    //Calculate Stop TIME (Start TIME + Shift Length TIME)
    IF  OEE_SP.Length.CurrentTime.wDay = 0 THEN			// When Length Day = 0, Stop Time Calculcation is Different because TimeStruct has a minimum of 1 for Days
    	_Year_Month_Day_TS[0].wHour 	 := OEE_SP.Length.CurrentTime.wHour;
    	_Year_Month_Day_TS[0].wMinute 	 := OEE_SP.Length.CurrentTime.wMinute;
    	_Stop_Time_DW 					 := ((_Start_Time_DW+_Year_Month_Day_DW[0])-_Year_Month_Day_DW[1]);	// Add Shift Length Time to Start Time and subtract Year/Month/Day = Stop Time
    	_Stop_Time_DT 					 := DWORD_TO_DT(_Stop_Time_DW);										// Convert Stop Time fron DWORD to DATE_AND_TIME format	
    	OEE_SP.Stop.CurrentTime 		 := DT_TO_SYSTEMTIME(_Stop_Time_DT);								// Convert Stop Time from DATE_AND_TIME format to TIMESTRUCT
    ELSE                                                                                
    	_Stop_Time_DW 					:= (_Start_Time_DW+_Length_Time_DW)-_Year_Month_Day_DW[1];	// Add Shift Length Time to Start Time and subtract Year/Month = Stop Time
    	_Stop_Time_DT 					:= DWORD_TO_DT(_Stop_Time_DW);								// Convert Stop Time fron DWORD to DATE_AND_TIME format
    	OEE_SP.Stop.CurrentTime 		:= DT_TO_SYSTEMTIME(_Stop_Time_DT);							// Convert Stop Time from DATE_AND_TIME format to TIMESTRUCT
    	OEE_SP.Stop.CurrentTime.wDay 	:= OEE_SP.Stop.CurrentTime.wDay + 1;
    END_IF
	
	IF NOT OEE_SP.Break_Active AND OEE_SP.Active THEN
		_fb_MachinePerfomance(Perf := OEE_SP.MachinePerformance, Control := Control, Data_Reset := _Mach_Perf_Reset);
	END_IF
    //--------------------------------------------------------Availability---------------------------------------------------------
    
    //Calculate total time the machine has been avaliable to run (i.e. operators not on a break)
    IF  OEE_SP.Active AND NOT OEE_SP.Break_Active AND Control.SystemTime.SecondPulse THEN;
    	OEE_SP.Production_Seconds := OEE_SP.Production_Seconds + 1;
    END_IF
    _Production_Time_T := REAL_TO_TIME(OEE_SP.Production_Seconds)*1000;
    _Production_Time_DT := TIME_TO_DT(_Production_Time_T);
    _Production_Time_TS := DT_TO_SYSTEMTIME(_Production_Time_DT);
    IF OEE_SP.Production_Seconds < 86400 THEN
    	OEE_SP.Production_Time.CurrentTime := _Production_Time_TS;
    	OEE_SP.Production_Time.CurrentTime.wDay := 0;
    ELSE
    	OEE_SP.Production_Time.CurrentTime := _Production_Time_TS;
    	OEE_SP.Production_Time.CurrentTime.wDay := _Production_Time_TS.wDay-1;
    END_IF	
    
    //Calculate the time the machine has been producing
    IF OEE_SP.Active AND NOT OEE_SP.Break_Active AND Control.SystemTime.SecondPulse AND (Control.PackMLState.Execute OR Control.PackMLState.Suspended OR Control.PackMLState.Suspending OR Control.PackMLState.UnSuspending) THEN;
    	OEE_SP.Operating_Seconds := OEE_SP.Operating_Seconds + 1;
    END_IF
    
    _Operating_Time_T := REAL_TO_TIME(OEE_SP.Operating_Seconds)*1000;
    _Operating_Time_DT := TIME_TO_DT(_Operating_Time_T);
    _Operating_Time_TS := DT_TO_SYSTEMTIME(_Operating_Time_DT);
    IF OEE_SP.Operating_Seconds < 86400 THEN
    	OEE_SP.Operating_Time.CurrentTime := (_Operating_Time_TS);
    	OEE_SP.Operating_Time.CurrentTime.wDay := 0;
    ELSE
    	OEE_SP.Operating_Time.CurrentTime := (_Operating_Time_TS);
    	OEE_SP.Operating_Time.CurrentTime.wDay := _Operating_Time_TS.wDay-1;
    END_IF
    
    //Calculate Break Time
    IF OEE_SP.Active AND OEE_SP.Break_Active AND Control.SystemTime.SecondPulse THEN;
    	OEE_SP.Break_Seconds := OEE_SP.Break_Seconds + 1; 
    END_IF
    _Break_Time_T := LREAL_TO_TIME(OEE_SP.Break_Seconds)*1000;
    _Break_Time_DT := TIME_TO_DT(_Break_Time_T);
    _Break_Time_TS := DT_TO_SYSTEMTIME(_Break_Time_DT);
    IF OEE_SP.Break_Seconds < 86400 THEN
    	OEE_SP.Break_Time.CurrentTime := (_Break_Time_TS);
    	OEE_SP.Break_Time.CurrentTime.wDay := 0;
    ELSE
    	OEE_SP.Break_Time.CurrentTime := (_Break_Time_TS);
    	OEE_SP.Break_Time.CurrentTime.wDay := _Break_Time_TS.wDay-1;
    END_IF
     
    //Calculate Avaliability
    IF (OEE_SP.Operating_Seconds > 0 AND OEE_SP.Production_Seconds > 0.0) AND Control.SystemTime.SecondPulse THEN;
    	OEE_SP.Availability := ((OEE_SP.Operating_Seconds/ F_CheckDivReal(OEE_SP.Production_Seconds))*100);
    ELSIF (OEE_SP.Operating_Seconds <= 0 OR OEE_SP.Production_Seconds <= 0.0) THEN;
    	OEE_SP.Availability := 0.0;
    END_IF
    
    //--------------------------------------------------------Performance---------------------------------------------------------
    
    //Calculate Performance
    IF (OEE_SP.TotalPieces > 0 AND OEE_SP.Operating_Seconds > 0.0 AND OEE_SP.TargetRate > 0.0) AND Control.SystemTime.SecondPulse  THEN;
    	OEE_SP.Performance := DINT_TO_REAL(OEE_SP.TotalPieces)/OEE_SP.Operating_Seconds/(F_CheckDivReal(OEE_SP.TargetRate/60))*100;
    ELSIF ((OEE_SP.TotalPieces <= 0) OR (OEE_SP.Operating_Seconds <= 0.0) OR (OEE_SP.TargetRate <= 0.0)) THEN;
    	OEE_SP.Performance := 0;
    ELSIF OEE_SP.Performance > 100.0 THEN;
    	OEE_SP.Performance := 100;
    END_IF
    
    //--------------------------------------------------------Quality---------------------------------------------------------
    
    //Calculate Quality
    IF (OEE_SP.GoodPieces > 0 AND OEE_SP.TotalPieces > 0) AND Control.SystemTime.SecondPulse  THEN;
    	OEE_SP.Quality := DINT_TO_REAL(OEE_SP.GoodPieces)/DINT_TO_REAL(F_CheckDivDint(OEE_SP.TotalPieces))*100;
    ELSIF (OEE_SP.GoodPieces <= 0 OR OEE_SP.TotalPieces <= 0) THEN;
    	OEE_SP.Quality := 0.0;
    END_IF
    //--------------------------------------------------------------OEE-----------------------------------------------------------------
    
    //Calculate OEE 
    IF Control.SystemTime.SecondPulse THEN
    OEE_SP.OEE := ((OEE_SP.Availability/100) * (OEE_SP.Performance/100) * (OEE_SP.Quality/100)) *100;
    IF OEE_SP.OEE >100.0 THEN
    	OEE_SP.OEE:=100;
    END_IF
    END_IF
    //--------------------------------------------------------Supply Availability---------------------------------------------------------
    
    //Calculate Infeed Supply
    IF (OEE_SP.Operating_Seconds > 0 AND OEE_SP.Production_Seconds > 0.0) AND Control.SystemTime.SecondPulse  THEN;
    	OEE_SP.SupplyAvaliability := ((OEE_SP.Operating_Seconds-(OEE_SP.SupplyDownTime_Seconds))/F_CheckDivReal(OEE_SP.Operating_Seconds)*100);
    ELSIF (OEE_SP.Operating_Seconds <= 0 OR OEE_SP.Production_Seconds <= 0.0) THEN;
    	OEE_SP.SupplyAvaliability := 0.0;
    END_IF
    //--------------------------------------------------------Outfeed Availability---------------------------------------------------------
    //Calculate Outfeed Availability
    IF (OEE_SP.Operating_Seconds > 0 AND OEE_SP.Production_Seconds > 0.0) AND Control.SystemTime.SecondPulse  THEN;
    	OEE_SP.OutfeedAvaliability := ((OEE_SP.Operating_Seconds-(OEE_SP.OutfeedDownTime_Seconds))/F_CheckDivReal(OEE_SP.Operating_Seconds)*100);
    ELSIF (OEE_SP.Operating_Seconds <= 0 OR OEE_SP.Production_Seconds <= 0.0) THEN;
    	OEE_SP.OutfeedAvaliability := 0.0;
    END_IF
    //--------------------------------------------------------Total Pieces---------------------------------------------------------
    OEE_SP.TotalPieces := (OEE_SP.GoodPieces + OEE_SP.RejectPieces);
    OEE.Outputs.Availability := OEE_SP.Availability;
    OEE.Outputs.Performance := OEE_SP.Performance;
    OEE.Outputs.Quality:= OEE_SP.Quality;
    OEE.Outputs.OEE:= OEE_SP.OEE;
	
	 //--------------------------------------------------------Active Shift---------------------------------------------------------
    _Current_Time_DT := SYSTEMTIME_TO_DT(_Current_Time.CurrentTime);
    _Current_Time_DW	:=DT_TO_DWORD(_Current_Time_DT);
    
    IF ((_Current_Time_DW > _Start_Time_DW) AND (_Current_Time_DW <= _Stop_Time_DW)) THEN //OR (REAL_TO_UDINT(OEE_SP.Production_Seconds) < (_Stop_Time_DW - _Start_Time_DW)) THEN
    	OEE.Outputs.Active := TRUE;
    	OEE_SP.Active := TRUE;
    ELSE 
    	OEE.Outputs.Active := FALSE;
    	OEE_SP.Active := FALSE;
    END_IF

	IF OEE.Inputs.Break_Active AND OEE.Outputs.Active THEN
		OEE_SP.Break_Active:=TRUE;
	ELSE 
		OEE_SP.Break_Active:=FALSE;
	END_IF
	
	OEE_SP.StateCurrent := Control.PackMLState.CurrentState;

END_FUNCTION_BLOCK

// Objects/FB_PML_V4_01/FB_PackML
FUNCTION_BLOCK FINAL FB_PackML
VAR_IN_OUT
	PackML							: ST_PMLData;
	Control							: ST_System;
END_VAR
VAR
	_Cfg_ModeTransitions			: ARRAY[0..9, 0..31] OF BOOL;
	_Index							: INT;
	_LastState						: DINT;
	_LastUnit						: DINT;
	_MessageClearPointer			: INT;
	_WarningRefreshPointer			: INT;
	_WarningRefresh					: F_TRIG;
END_VAR
VAR CONSTANT
	_MaxModeLength					: INT := 7;
	_MaxStateLength					: INT := 17;
END_VAR
VAR PERSISTENT
	_LS_H_IndicatorMatrix				: ARRAY[0..31] OF DINT :=[1032,33792,1032,361504,66784,361504,198690,67616,1028,1028,1032,99360,1216,82984,295936,1032,1028];
	_PB_IndicatorMatrix					: ARRAY[0..31] OF DINT :=[0,256,32768,0,32768,32768,32768,16384,0,256,0,0,32768,32768,16384,32768,256,0];			
	_LS_H_IndicatorDescription			: ARRAY[0..31] OF STRING(40) := ['','Alarm','Abnormal Stop','Controlled Stop','','Alert','Starved Upstream','Blocked Downstream','','','Low Material','Material Exhausted','','','Alert','Alarm','Starting / Restarting','','','','','','','','','','','','',''];		
	_PB_IndicatorDescription			: ARRAY[0..31] OF STRING(40) := ['','','','','','','','','Ready to Reset','','','','','','Ready to Start','Running','','','','','','','','','','','','','','','',''];		
END_VAR

M_Administration();
M_Commands();
M_Indicators();
M_ModeControl();
M_SafetyBreach();
M_StateMapping();
M_StateTransitions();
M_TransitionCounts();

METHOD PRIVATE M_Administration
VAR_INPUT
END_VAR
VAR_INST
	_index					: INT;
END_VAR
IF PackML.Status.UnitModeCurrent > _maxModeLength THEN
	PackML.Control.UnitMode := 0;
	PackML.Status.UnitModeCurrent := 0;
END_IF

//Time spent in Mode
//The elapsed time the machine has spent in that mode since it entered that mode.  Array index is equal to designation of the mode.
IF PackML.Status.UnitModeChangeInProcess THEN
	PackML.Admin.ModeCurrentTime[PackML.Status.UnitModeCurrent] := 0;
END_IF
IF Control.SystemTime.SecondPulse THEN
	PackML.Admin.ModeCurrentTime[PackML.Status.UnitModeCurrent] := PackML.Admin.ModeCurrentTime[PackML.Status.UnitModeCurrent] + 1;
	IF PackML.Admin.ModeCurrentTime[PackML.Status.UnitModeCurrent] < 0 THEN
		PackML.Admin.ModeCurrentTime[PackML.Status.UnitModeCurrent] := 0;
	END_IF
	IF PackML.Admin.ResetTimerCounters THEN
		FOR _index := 0 TO _maxModeLength DO
			PackML.Admin.ModeCurrentTime[_index] := 0;
		END_FOR
	END_IF
END_IF

//Cumulative TIME In Each Mode
//The cumulative elapsed time the machine has spent in each mode since it’s timers and counters were reset.  
IF Control.SystemTime.SecondPulse THEN
	PackML.Admin.ModeCummulativeTime[PackML.Status.UnitModeCurrent] := PackML.Admin.ModeCummulativeTime[PackML.Status.UnitModeCurrent] + 1;
	IF PackML.Admin.ModeCummulativeTime[PackML.Status.UnitModeCurrent] < 0 THEN
		PackML.Admin.ModeCummulativeTime[PackML.Status.UnitModeCurrent] := 0;
	END_IF
	IF PackML.Admin.ResetTimerCounters THEN
		FOR _index := 0 TO _maxModeLength DO
			PackML.Admin.ModeCummulativeTime[_index] := 0;
		END_FOR
	END_IF
END_IF

//TIME spent in State
//The elapsed time the machine has spent in that State since it entered that State.  Array index is equal to designation of the mode.
IF PackML.Status.StateChangeInProgress THEN
	PackML.Admin.StateCurrentTime[PackML.Status.UnitModeCurrent,PackML.Status.StateCurrent] := 0;
END_IF
IF Control.SystemTime.SecondPulse THEN
	PackML.Admin.StateCurrentTime[PackML.Status.UnitModeCurrent,PackML.Status.StateCurrent] := PackML.Admin.StateCurrentTime[PackML.Status.UnitModeCurrent,PackML.Status.StateCurrent] + 1;
	IF PackML.Admin.StateCurrentTime[PackML.Status.UnitModeCurrent,PackML.Status.StateCurrent] < 0 THEN
		PackML.Admin.StateCurrentTime[PackML.Status.UnitModeCurrent,PackML.Status.StateCurrent] := 0;
	END_IF
	IF PackML.Admin.ResetTimerCounters THEN
		FOR _index := 0 TO _maxStateLength DO
			PackML.Admin.StateCurrentTime[PackML.Status.UnitModeCurrent,_index] := 0;
		END_FOR
	END_IF
END_IF

//Cumulative Time In Each Mode
//The cumulative elapsed time the machine has spent in each mode since it’s timers and counters were reset.  
IF Control.SystemTime.SecondPulse THEN
	PackML.Admin.StateCummulativeTime[PackML.Status.UnitModeCurrent,PackML.Status.StateCurrent] := PackML.Admin.StateCummulativeTime[PackML.Status.UnitModeCurrent,PackML.Status.StateCurrent] + 1;
	IF PackML.Admin.StateCummulativeTime[PackML.Status.UnitModeCurrent,PackML.Status.StateCurrent] < 0 THEN
		PackML.Admin.StateCummulativeTime[PackML.Status.UnitModeCurrent,PackML.Status.StateCurrent] := 0;
	END_IF
	IF PackML.Admin.ResetTimerCounters THEN
		FOR _index := 0 TO _maxStateLength DO
			PackML.Admin.StateCummulativeTime[PackML.Status.UnitModeCurrent,_index] := 0;
		END_FOR
	END_IF
END_IF
END_METHOD

METHOD PRIVATE M_Commands
VAR_INPUT
END_VAR
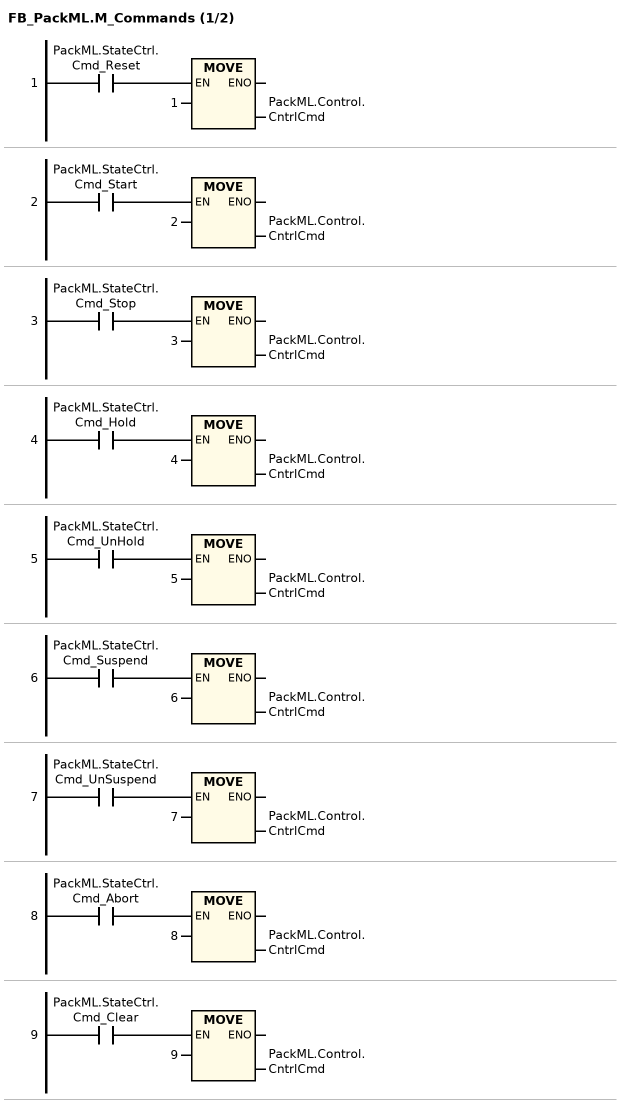
// NETWORK 1
IF PackML.StateCtrl.Cmd_Reset THEN PackML.Control.CntrlCmd := 1; END_IF

// NETWORK 2
IF PackML.StateCtrl.Cmd_Start THEN PackML.Control.CntrlCmd := 2; END_IF

// NETWORK 3
IF PackML.StateCtrl.Cmd_Stop THEN PackML.Control.CntrlCmd := 3; END_IF

// NETWORK 4
IF PackML.StateCtrl.Cmd_Hold THEN PackML.Control.CntrlCmd := 4; END_IF

// NETWORK 5
IF PackML.StateCtrl.Cmd_UnHold THEN PackML.Control.CntrlCmd := 5; END_IF

// NETWORK 6
IF PackML.StateCtrl.Cmd_Suspend THEN PackML.Control.CntrlCmd := 6; END_IF

// NETWORK 7
IF PackML.StateCtrl.Cmd_UnSuspend THEN PackML.Control.CntrlCmd := 7; END_IF

// NETWORK 8
IF PackML.StateCtrl.Cmd_Abort THEN PackML.Control.CntrlCmd := 8; END_IF

// NETWORK 9
IF PackML.StateCtrl.Cmd_Clear THEN PackML.Control.CntrlCmd := 9; END_IF

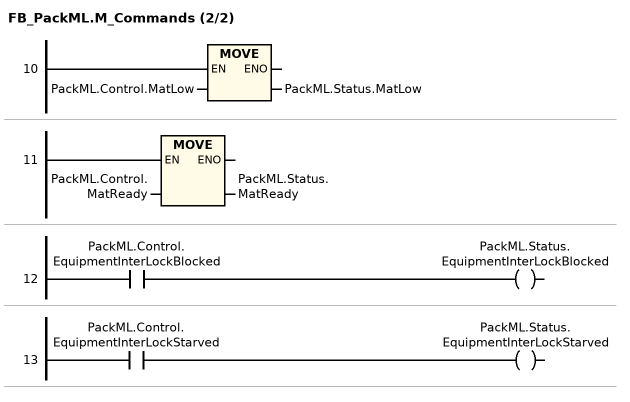
// NETWORK 10
PackML.Status.MatLow := PackML.Control.MatLow;

// NETWORK 11
PackML.Status.MatReady := PackML.Control.MatReady;

// NETWORK 12
PackML.Status.EquipmentInterLockBlocked := PackML.Control.EquipmentInterLockBlocked;

// NETWORK 13
PackML.Status.EquipmentInterLockStarved := PackML.Control.EquipmentInterLockStarved;
END_METHOD

METHOD PRIVATE M_Indicators
VAR_INST
	_i 		: DINT;
	_f_trig	: F_TRIG;
	_r_trig	: R_TRIG;
	k : bool;
END_VAR
PackML.Indicator.LS_H_Output := _LS_H_IndicatorMatrix[PackML.Status.StateCurrent];

//Red Lamp
IF PackML.Indicator.LS_H_Output.0 THEN
	PackML.Indicator.RedLamp := Control.SystemTime.PulseFlash;
ELSIF PackML.Indicator.LS_H_Output.1 AND Control.Outputs.Alarm THEN
	PackML.Indicator.RedLamp := Control.SystemTime.FastFlash;
ELSIF PackML.Indicator.LS_H_Output.2 THEN
	PackML.Indicator.RedLamp := Control.SystemTime.SlowFlash;
ELSIF PackML.Indicator.LS_H_Output.3 THEN
	PackML.Indicator.RedLamp := TRUE;
ELSE
	PackML.Indicator.RedLamp := FALSE;
END_IF

//Amber Lamp
IF PackML.Indicator.LS_H_Output.4 THEN
	PackML.Indicator.AmberLamp := Control.SystemTime.PulseFlash;
ELSIF PackML.Indicator.LS_H_Output.5 AND Control.Outputs.Alert THEN
	PackML.Indicator.AmberLamp := Control.SystemTime.FastFlash;
ELSIF PackML.Indicator.LS_H_Output.6 THEN
	PackML.Indicator.AmberLamp := Control.SystemTime.SlowFlash;
ELSIF PackML.Indicator.LS_H_Output.7 THEN
	PackML.Indicator.AmberLamp := TRUE;
ELSE
	PackML.Indicator.AmberLamp := FALSE;
END_IF

//Blue Lamp
IF PackML.Indicator.LS_H_Output.8 THEN
	PackML.Indicator.BlueLamp := Control.SystemTime.PulseFlash;
ELSIF PackML.Indicator.LS_H_Output.9 THEN
	PackML.Indicator.BlueLamp := Control.SystemTime.FastFlash;
ELSIF PackML.Indicator.LS_H_Output.10 THEN
	FOR	_i := 0 TO SIZEOF(Packml.Status.MatLow) BY 1 DO
		IF Packml.Status.MatLow[_i] THEN
			PackML.Indicator.BlueLamp := Control.SystemTime.SlowFlash;
			EXIT;
		END_IF
	END_FOR
ELSIF PackML.Indicator.LS_H_Output.11 THEN
	FOR	_i := 0 TO SIZEOF(Packml.Status.MatReady) BY 1 DO
		_f_trig(CLK:= Packml.Status.MatReady[_i]);
		IF _f_trig.Q THEN
			PackML.Indicator.BlueLamp := TRUE;
			EXIT;
		END_IF
		_r_trig(CLK:= Packml.Status.MatReady[_i]);
		IF _r_trig.Q THEN
			PackML.Indicator.BlueLamp := FALSE;
			EXIT;
		END_IF
	END_FOR
ELSE
	PackML.Indicator.BlueLamp := FALSE;
END_IF

//Green Lamp
IF PackML.Indicator.LS_H_Output.12 THEN
	PackML.Indicator.GreenLamp := Control.SystemTime.PulseFlash;
ELSIF PackML.Indicator.LS_H_Output.13 THEN
	PackML.Indicator.GreenLamp := Control.SystemTime.FastFlash;
ELSIF PackML.Indicator.LS_H_Output.14 THEN
	PackML.Indicator.GreenLamp := Control.SystemTime.SlowFlash;
ELSIF PackML.Indicator.LS_H_Output.15 THEN
	PackML.Indicator.GreenLamp := TRUE;
ELSE
	PackML.Indicator.GreenLamp := FALSE;
END_IF

//Horn
IF PackML.Indicator.LS_H_Output.16 AND Control.Outputs.Alert THEN
	PackML.Indicator.Horn := Control.SystemTime.PulseFlash;
ELSIF PackML.Indicator.LS_H_Output.17 AND Control.Outputs.Alarm THEN
	PackML.Indicator.Horn := Control.SystemTime.FastFlash;
ELSIF PackML.Indicator.LS_H_Output.18 THEN
	PackML.Indicator.Horn := Control.SystemTime.SlowFlash;
ELSIF PackML.Indicator.LS_H_Output.19 THEN
	PackML.Indicator.Horn := TRUE;
ELSE
	PackML.Indicator.Horn := FALSE;
END_IF

PackML.Indicator.PB_Output := _PB_IndicatorMatrix[PackML.Status.StateCurrent];

//Red Button
IF PackML.Indicator.PB_Output.0 THEN
	PackML.Indicator.RedButton := Control.SystemTime.PulseFlash;
ELSIF PackML.Indicator.PB_Output.1 THEN
	PackML.Indicator.RedButton := Control.SystemTime.FastFlash;
ELSIF PackML.Indicator.PB_Output.2 THEN
	PackML.Indicator.RedButton := Control.SystemTime.SlowFlash;
ELSIF PackML.Indicator.PB_Output.3 THEN
	PackML.Indicator.RedButton := TRUE;
ELSE
	PackML.Indicator.RedButton := FALSE;
END_IF

//Amber Button
IF PackML.Indicator.PB_Output.4 THEN
	PackML.Indicator.AmberButton := Control.SystemTime.PulseFlash;
ELSIF PackML.Indicator.PB_Output.5 THEN
	PackML.Indicator.AmberButton := Control.SystemTime.FastFlash;
ELSIF PackML.Indicator.PB_Output.6 THEN
	PackML.Indicator.AmberButton := Control.SystemTime.SlowFlash;
ELSIF PackML.Indicator.PB_Output.7 THEN
	PackML.Indicator.AmberButton := TRUE;
ELSE
	PackML.Indicator.AmberButton := FALSE;
END_IF

//Blue Button
IF PackML.Indicator.PB_Output.8 THEN
	PackML.Indicator.BlueButton := Control.SystemTime.PulseFlash;
ELSIF PackML.Indicator.PB_Output.9 THEN
	PackML.Indicator.BlueButton := Control.SystemTime.FastFlash;
ELSIF PackML.Indicator.PB_Output.10 THEN
	PackML.Indicator.BlueButton := Control.SystemTime.SlowFlash;
ELSIF PackML.Indicator.PB_Output.11 THEN
	PackML.Indicator.BlueButton := TRUE;
ELSE
	PackML.Indicator.BlueButton := FALSE;
END_IF

//Green Button
IF PackML.Indicator.PB_Output.12 THEN
	PackML.Indicator.GreenButton := Control.SystemTime.PulseFlash;
ELSIF PackML.Indicator.PB_Output.13 THEN
	PackML.Indicator.GreenButton := Control.SystemTime.FastFlash;
ELSIF PackML.Indicator.PB_Output.14 THEN
	PackML.Indicator.GreenButton := Control.SystemTime.SlowFlash;
ELSIF PackML.Indicator.PB_Output.15 THEN
	PackML.Indicator.GreenButton := TRUE;
ELSE
	PackML.Indicator.GreenButton := FALSE;
END_IF
END_METHOD

METHOD PRIVATE M_ModeControl
VAR_INPUT
END_VAR
VAR_INST
END_VAR
IF Control.SystemTime.FirstCycle THEN
	FOR _index := 0 TO 9 BY 1 DO
		_cfg_ModeTransitions[_index,2] := TRUE;
		_cfg_ModeTransitions[_index,9] := TRUE;
	END_FOR
END_IF

IF PackML.Control.UnitMode >= 1 AND PackML.Control.UnitMode <= 32 AND (PackML.Control.UnitMode <> PackML.Status.UnitModeCurrent) THEN
	IF _cfg_ModeTransitions[PackML.Status.UnitModeCurrent,PackML.Status.StateCurrent] AND _cfg_ModeTransitions[PackML.Control.UnitMode,PackML.Status.StateCurrent] THEN
		PackML.Status.UnitModeCurrent := PackML.Control.UnitMode;
	END_IF
	PackML.Control.UnitModeChangeRequest := TRUE;
	PackML.Status.UnitModeRequested := TRUE;
ELSE
	PackML.Control.UnitModeChangeRequest := FALSE;
	PackML.Status.UnitModeRequested := FALSE;
END_IF
END_METHOD

METHOD PRIVATE M_SafetyBreach
VAR_INPUT
END_VAR
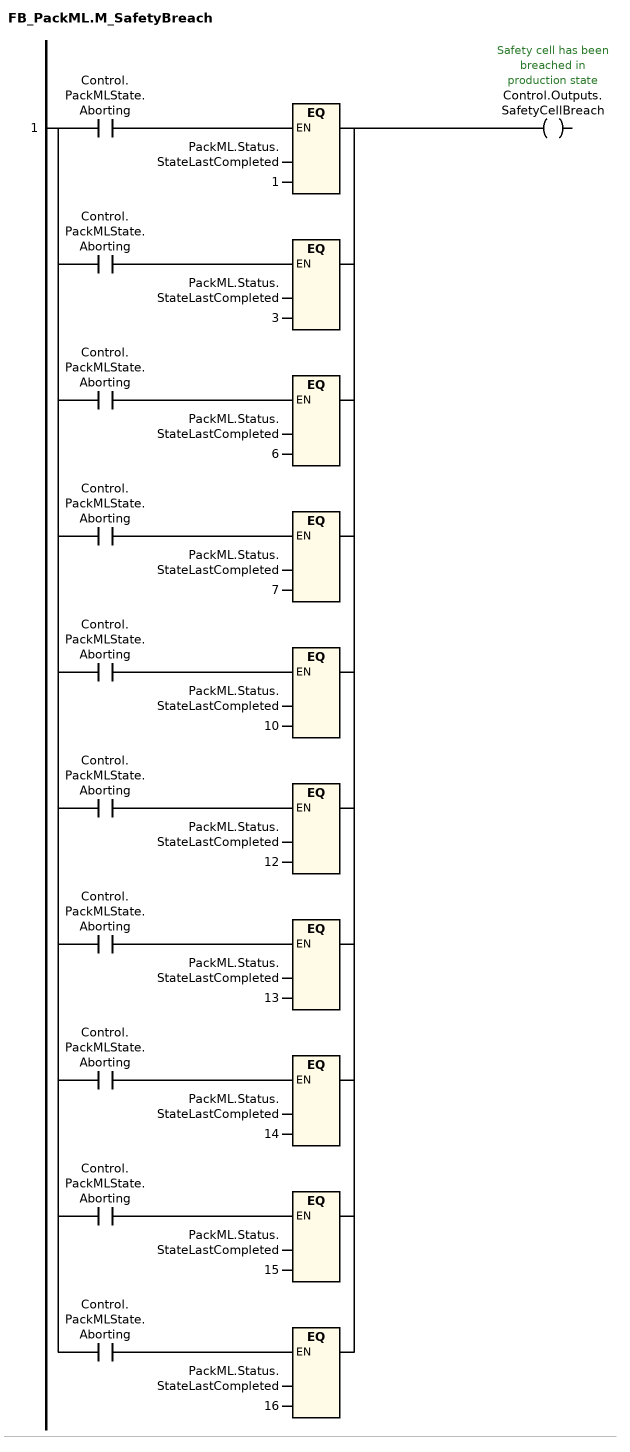
// NETWORK 1
//   PackML.Status.StateLastCompleted: Last Completed State
//   Control.Outputs.SafetyCellBreach: Safety cell has been breached in production state
Control.Outputs.SafetyCellBreach := Control.PackMLState.Aborting AND PackML.Status.StateLastCompleted = 1 OR Control.PackMLState.Aborting AND PackML.Status.StateLastCompleted = 3 OR Control.PackMLState.Aborting AND PackML.Status.StateLastCompleted = 6 OR Control.PackMLState.Aborting AND PackML.Status.StateLastCompleted = 7 OR Control.PackMLState.Aborting AND PackML.Status.StateLastCompleted = 10 OR Control.PackMLState.Aborting AND PackML.Status.StateLastCompleted = 12 OR Control.PackMLState.Aborting AND PackML.Status.StateLastCompleted = 13 OR Control.PackMLState.Aborting AND PackML.Status.StateLastCompleted = 14 OR Control.PackMLState.Aborting AND PackML.Status.StateLastCompleted = 15 OR Control.PackMLState.Aborting AND PackML.Status.StateLastCompleted = 16;
END_METHOD

METHOD PRIVATE M_StateMapping
VAR_INPUT
END_VAR
VAR_INST
END_VAR
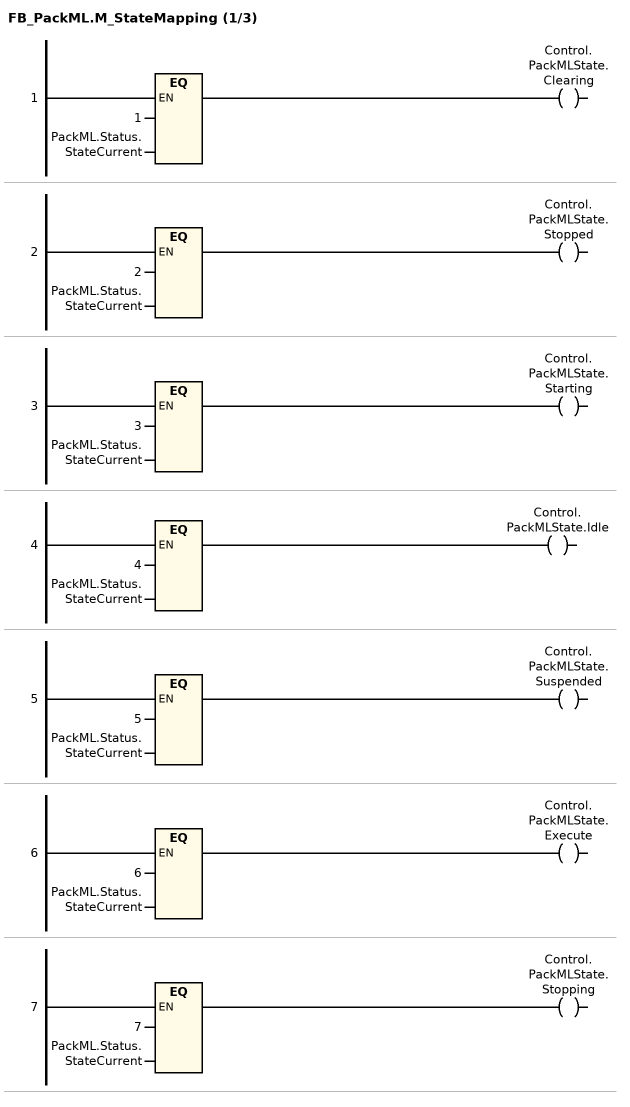
// NETWORK 1
//   PackML.Status.StateCurrent: Current State Number
Control.PackMLState.Clearing := 1 = PackML.Status.StateCurrent;

// NETWORK 2
//   PackML.Status.StateCurrent: Current State Number
Control.PackMLState.Stopped := 2 = PackML.Status.StateCurrent;

// NETWORK 3
//   PackML.Status.StateCurrent: Current State Number
Control.PackMLState.Starting := 3 = PackML.Status.StateCurrent;

// NETWORK 4
//   PackML.Status.StateCurrent: Current State Number
Control.PackMLState.Idle := 4 = PackML.Status.StateCurrent;

// NETWORK 5
//   PackML.Status.StateCurrent: Current State Number
Control.PackMLState.Suspended := 5 = PackML.Status.StateCurrent;

// NETWORK 6
//   PackML.Status.StateCurrent: Current State Number
Control.PackMLState.Execute := 6 = PackML.Status.StateCurrent;

// NETWORK 7
//   PackML.Status.StateCurrent: Current State Number
Control.PackMLState.Stopping := 7 = PackML.Status.StateCurrent;

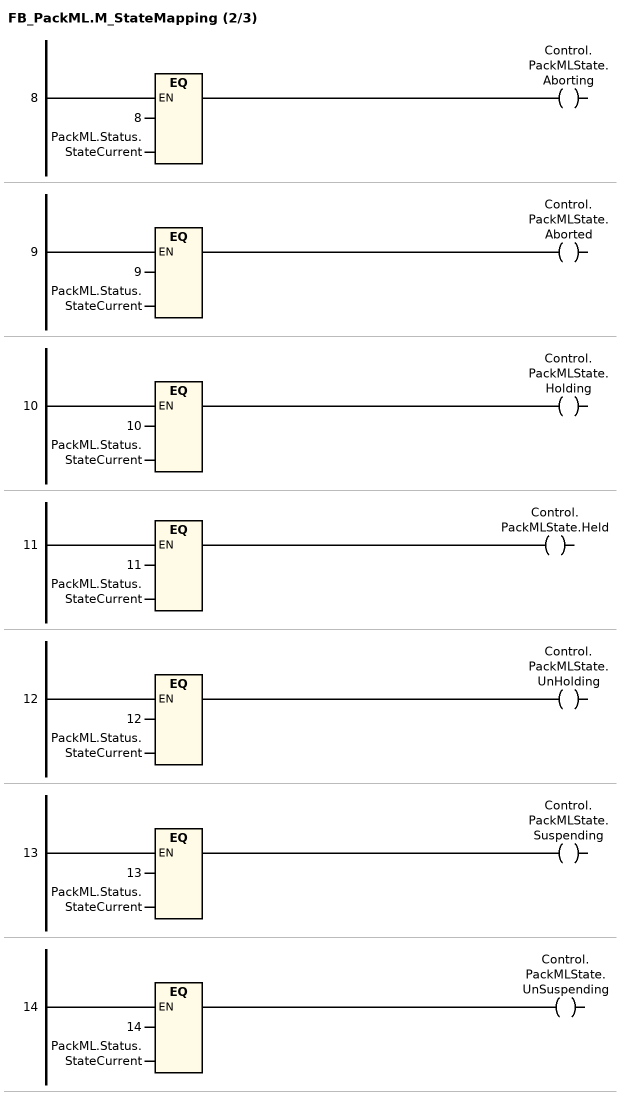
// NETWORK 8
//   PackML.Status.StateCurrent: Current State Number
Control.PackMLState.Aborting := 8 = PackML.Status.StateCurrent;

// NETWORK 9
//   PackML.Status.StateCurrent: Current State Number
Control.PackMLState.Aborted := 9 = PackML.Status.StateCurrent;

// NETWORK 10
//   PackML.Status.StateCurrent: Current State Number
Control.PackMLState.Holding := 10 = PackML.Status.StateCurrent;

// NETWORK 11
//   PackML.Status.StateCurrent: Current State Number
Control.PackMLState.Held := 11 = PackML.Status.StateCurrent;

// NETWORK 12
//   PackML.Status.StateCurrent: Current State Number
Control.PackMLState.UnHolding := 12 = PackML.Status.StateCurrent;

// NETWORK 13
//   PackML.Status.StateCurrent: Current State Number
Control.PackMLState.Suspending := 13 = PackML.Status.StateCurrent;

// NETWORK 14
//   PackML.Status.StateCurrent: Current State Number
Control.PackMLState.UnSuspending := 14 = PackML.Status.StateCurrent;

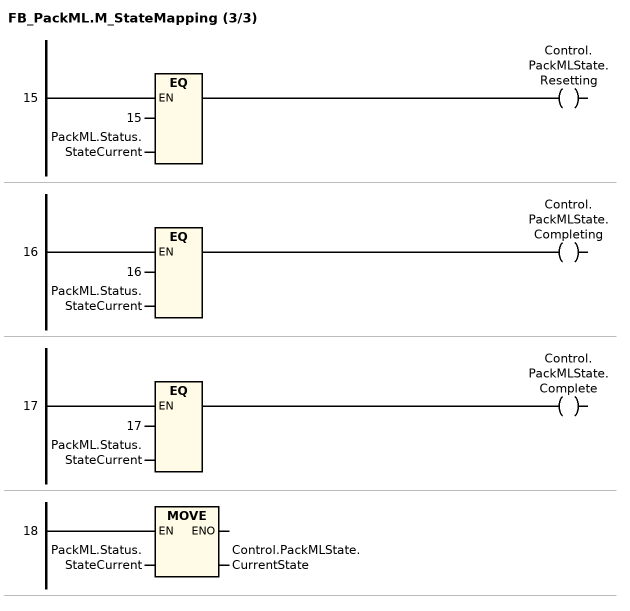
// NETWORK 15
//   PackML.Status.StateCurrent: Current State Number
Control.PackMLState.Resetting := 15 = PackML.Status.StateCurrent;

// NETWORK 16
//   PackML.Status.StateCurrent: Current State Number
Control.PackMLState.Completing := 16 = PackML.Status.StateCurrent;

// NETWORK 17
//   PackML.Status.StateCurrent: Current State Number
Control.PackMLState.Complete := 17 = PackML.Status.StateCurrent;

// NETWORK 18
//   PackML.Status.StateCurrent: Current State Number
Control.PackMLState.CurrentState := PackML.Status.StateCurrent;
END_METHOD

METHOD PRIVATE M_StateTransitions
VAR_INPUT
END_VAR
VAR_INST
END_VAR
//Clearing - 1
IF Control.PackMLState.Aborted AND PackML.StateCtrl.Cmd_Clear THEN
	PackML.Control.State := 1;
	PackML.Status.StateLastCompleted := PackML.Status.StateCurrent;
	PackML.Status.StateCurrent := PackML.Control.State;
END_IF

//Stopped - 2
IF Control.PackMLState.Stopping OR Control.PackMLState.Clearing THEN
	PackML.Control.State := 2;
	IF PackML.Control.StateChangeRequest THEN
		PackML.Status.StateLastCompleted := PackML.Status.StateCurrent;
		PackML.Status.StateCurrent := PackML.Control.State;
	END_IF
END_IF

//Starting - 3
IF Control.PackMLState.Idle AND PackML.StateCtrl.Cmd_Start THEN
	PackML.Control.State := 3;
	PackML.Status.StateLastCompleted := PackML.Status.StateCurrent;
	PackML.Status.StateCurrent := PackML.Control.State;
END_IF

//Idle - 4
IF Control.PackMLState.Resetting THEN
	PackML.Control.State := 4;
	IF PackML.Control.StateChangeRequest THEN
		PackML.Status.StateLastCompleted := PackML.Status.StateCurrent;
		PackML.Status.StateCurrent := PackML.Control.State;
	END_IF
END_IF

//Suspended - 5
IF Control.PackMLState.Suspending THEN
	PackML.Control.State := 5;
	IF PackML.Control.StateChangeRequest THEN
		PackML.Status.StateLastCompleted := PackML.Status.StateCurrent;
		PackML.Status.StateCurrent := PackML.Control.State;
	END_IF
END_IF

//Execute - 6
IF Control.PackMLState.Starting OR Control.PackMLState.UnHolding OR Control.PackMLState.UnSuspending THEN
	PackML.Control.State := 6;
	IF PackML.Control.StateChangeRequest THEN
		PackML.Status.StateLastCompleted := PackML.Status.StateCurrent;
		PackML.Status.StateCurrent := PackML.Control.State;
	END_IF
END_IF

//Stopping - 7
IF (Control.PackMLState.Resetting 
OR Control.PackMLState.Idle 
OR Control.PackMLState.Starting 
OR Control.PackMLState.Execute 
OR Control.PackMLState.Holding 
OR Control.PackMLState.Held 
OR Control.PackMLState.UnHolding 
OR Control.PackMLState.Suspending
OR Control.PackMLState.Suspended
OR Control.PackMLState.UnSuspending 
OR Control.PackMLState.Completing 
OR Control.PackMLState.Clearing 
OR Control.PackMLState.Complete) 
AND PackML.StateCtrl.Cmd_Stop THEN
	PackML.Control.State := 7;
	PackML.Status.StateLastCompleted := PackML.Status.StateCurrent;
	PackML.Status.StateCurrent := PackML.Control.State;
END_IF

//Aborting - 8
IF (NOT Control.PackMLState.Aborting AND NOT Control.PackMLState.Aborted AND PackML.StateCtrl.Cmd_Abort) 
OR (PackML.Control.State <= 0 OR PackML.Control.State >= 18) 
OR (PackML.Status.StateCurrent <= 0 OR PackML.Status.StateCurrent >= 18)  THEN
	PackML.Control.State := 8;
	PackML.Status.StateLastCompleted := PackML.Status.StateCurrent;
	PackML.Status.StateCurrent := PackML.Control.State;
END_IF

//Abort - 9
IF Control.PackMLState.Aborting THEN
	PackML.Control.State := 9;
	IF PackML.Control.StateChangeRequest THEN
		PackML.Status.StateLastCompleted := PackML.Status.StateCurrent;
		PackML.Status.StateCurrent := PackML.Control.State;
	END_IF
END_IF

//Holding - 10
IF Control.PackMLState.Execute AND PackML.StateCtrl.Cmd_Hold THEN
	PackML.Control.State := 10;
	PackML.Status.StateLastCompleted := PackML.Status.StateCurrent;
	PackML.Status.StateCurrent := PackML.Control.State;
END_IF

//Held - 11
IF Control.PackMLState.Holding THEN
	PackML.Control.State := 11;
	IF PackML.Control.StateChangeRequest THEN
		PackML.Status.StateLastCompleted := PackML.Status.StateCurrent;
		PackML.Status.StateCurrent := PackML.Control.State;
	END_IF
END_IF

//Unholding - 12
IF Control.PackMLState.Held AND PackML.StateCtrl.Cmd_UnHold THEN
	PackML.Control.State := 12;
	PackML.Status.StateLastCompleted := PackML.Status.StateCurrent;
	PackML.Status.StateCurrent := PackML.Control.State;
END_IF

//Suspending - 13
IF Control.PackMLState.Execute AND PackML.StateCtrl.Cmd_Suspend THEN
	PackML.Control.State := 13;
	PackML.Status.StateLastCompleted := PackML.Status.StateCurrent;
	PackML.Status.StateCurrent := PackML.Control.State;
END_IF

//UnSuspending - 14
IF Control.PackMLState.Suspended AND PackML.StateCtrl.Cmd_UnSuspend THEN
	PackML.Control.State := 14;
	PackML.Status.StateLastCompleted := PackML.Status.StateCurrent;
	PackML.Status.StateCurrent := PackML.Control.State;
END_IF

//Resetting - 15
IF (Control.PackMLState.Stopped 
OR Control.PackMLState.Complete)
AND PackML.StateCtrl.Cmd_Reset THEN
	PackML.Control.State := 15;
	PackML.Status.StateLastCompleted := PackML.Status.StateCurrent;
	PackML.Status.StateCurrent := PackML.Control.State;
END_IF

//Completing - 16
IF Control.PackMLState.Execute AND PackML.StateCtrl.Sts_Execute_SC THEN
	PackML.Control.State := 16;
	PackML.Status.StateLastCompleted := PackML.Status.StateCurrent;
	PackML.Status.StateCurrent := PackML.Control.State;
END_IF

//Complete - 17
IF Control.PackMLState.Completing THEN
	PackML.Control.State := 17;
	IF PackML.Control.StateChangeRequest THEN
		PackML.Status.StateLastCompleted := PackML.Status.StateCurrent;
		PackML.Status.StateCurrent := PackML.Control.State;
	END_IF
END_IF
END_METHOD

METHOD PRIVATE M_TransitionCounts
VAR_INPUT
END_VAR
VAR_INST
END_VAR
VAR_INST // added by the converter: edge detectors and wires of the graphical bodies
    _w1, _w2 : BOOL;
END_VAR
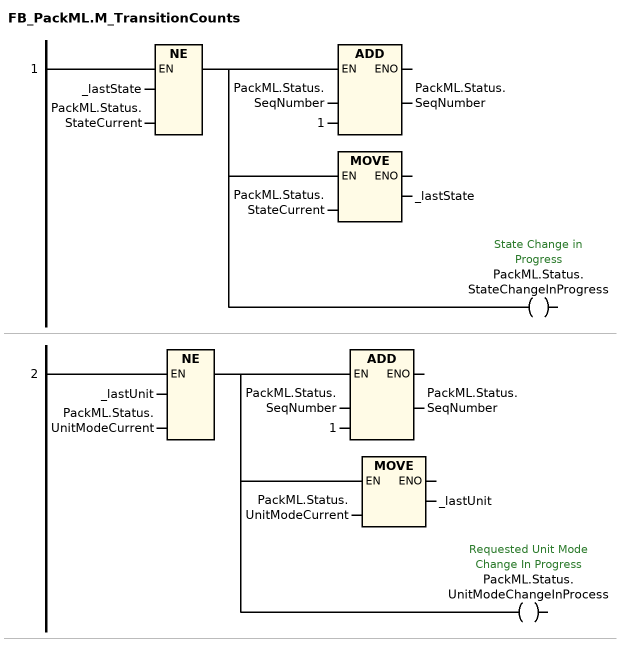
// NETWORK 1
//   PackML.Status.StateCurrent: Current State Number
//   PackML.Status.SeqNumber: Pack ML Sequence Number
//   PackML.Status.StateChangeInProgress: State Change in Progress
_w1 := _lastState <> PackML.Status.StateCurrent;
IF _w1 THEN PackML.Status.SeqNumber := PackML.Status.SeqNumber + 1; END_IF
IF _w1 THEN _lastState := PackML.Status.StateCurrent; END_IF
PackML.Status.StateChangeInProgress := _w1;

// NETWORK 2
//   PackML.Status.UnitModeCurrent: Unit Mode in current use
//   PackML.Status.SeqNumber: Pack ML Sequence Number
//   PackML.Status.UnitModeChangeInProcess: Requested Unit Mode Change In Progress
_w2 := _lastUnit <> PackML.Status.UnitModeCurrent;
IF _w2 THEN PackML.Status.SeqNumber := PackML.Status.SeqNumber + 1; END_IF
IF _w2 THEN _lastUnit := PackML.Status.UnitModeCurrent; END_IF
PackML.Status.UnitModeChangeInProcess := _w2;
END_METHOD

END_FUNCTION_BLOCK

// Objects/FB_Service_V3_00/FB_Service
FUNCTION_BLOCK FINAL FB_Service
VAR_IN_OUT
	Control				: ST_System;
END_VAR
VAR
	_ServiceDue			: BOOL;//Machine Service Due
	_Services			: SINT;//Service History Loop
	_ServiceReset		: BOOL;//Service Reset Selection
END_VAR
VAR PERSISTENT
	_LastBy				: STRING;// Last service done by
	_LastDate			: TIMESTRUCT;// Last service date
	_NextDueMonths		: REAL;// Next service due months
	_NextDueHours		: REAL;// Next service due hours
	_NextDueDate		: TIMESTRUCT;// Next service due date
	_IntervalMonths		: REAL := 12;// Service interval months
	_IntervalHours		: REAL := 20000;// Service interval hours
	_MachineHours		: REAL;// Service machine hours
	_HoursRemaining		: REAL;// Service hours remaining
	_History			: ARRAY[0..9,0..3] OF STRING(31);// Service history
END_VAR

// Update Machine Running Hours
IF (Control.PackMLState.Execute OR Control.PackMLState.Holding OR Control.PackMLState.UnHolding OR Control.PackMLState.Suspending OR Control.PackMLState.UnSuspending) AND Control.SystemTime.SecondPulse THEN
	// Increment machine running hours
	_MachineHours := _MachineHours + (1.00/3600.00);
	// Update Hours remaining until next service
	IF (_MachineHours < _NextDueHours) THEN _HoursRemaining := (_NextDueHours - _MachineHours); END_IF
	IF (_MachineHours >= _NextDueHours) THEN _HoursRemaining := 0; END_IF

END_IF

// Check If A Service Is Due
_ServiceDue := (_MachineHours > _NextDueHours) OR ((Control.SystemTime.CurrentTime.wYear >= _NextDueDate.wYear) AND (Control.SystemTime.CurrentTime.wMonth >= _NextDueDate.wMonth) AND (Control.SystemTime.CurrentTime.wDay >= _NextDueDate.wDay));

// Service Reset
IF _ServiceReset THEN
	// Update last service date
	_LastDate := Control.SystemTime.CurrentTime;
	
	// Update next service hours
	_NextDueHours := _MachineHours + _IntervalHours;
	_HoursRemaining := _NextDueHours - _MachineHours;
	
	// Calculate the next service due date
	_NextDueDate.wDay := Control.SystemTime.CurrentTime.wDay;
	_NextDueDate.wMonth := Control.SystemTime.CurrentTime.wMonth + REAL_TO_WORD(_IntervalMonths);
	_NextDueDate.wYear := Control.SystemTime.CurrentTime.wYear;
	
	// Check month overflow
	WHILE _NextDueDate.wMonth > 12 DO 
		_NextDueDate.wMonth := _NextDueDate.wMonth - 12;
		_NextDueDate.wYear := Control.SystemTime.CurrentTime.wYear + 1;
	END_WHILE
	
	//Service History
	FOR _Services :=8 TO 0 BY -1 DO
		_History[_Services+1,0] := _History[_Services,0];
		_History[_Services+1,1] := _History[_Services,1];
		_History[_Services+1,2] := _History[_Services,2];
		_History[_Services+1,3] := _History[_Services,3];
	END_FOR;
	_History[0,0] := _LastBy;
	_History[0,1] := TO_STRING(_MachineHours);
	_History[0,2] := SYSTEMTIME_TO_STRING(_LastDate);
	_History[0,3] := SYSTEMTIME_TO_STRING(_NextDueDate);
	_ServiceReset := FALSE;
END_IF

END_FUNCTION_BLOCK

// Objects/FB_Servo_V4_07/Helpers/F_ServoCheckWindow
FUNCTION F_ServoCheckWindow : BOOL
VAR_INPUT
	Unwind			: LREAL;
	Value			: LREAL;
	Target			: REAL;
	Tollerance		: REAL;
END_VAR
VAR
	UpperBound		: REAL;
	LowerBound		: REAL;
END_VAR

LowerBound := Target - Tollerance;
UpperBound := Target + Tollerance;

IF LowerBound >= 0 AND UpperBound <= Unwind THEN
	F_ServoCheckWindow := ((Value >= LowerBound) AND (Value <= UpperBound));
ELSIF LowerBound < 0 THEN
	F_ServoCheckWindow := (((Value >= (Unwind + LowerBound)) AND (Value <= Unwind)) OR (Value >= 0) AND (Value <= UpperBound));
ELSIF UpperBound > Unwind THEN
	F_ServoCheckWindow := (((Value >= LowerBound) AND (Value <= Unwind)) OR (Value >= 0) AND (Value <= (UpperBound - Unwind)));
ELSE
	F_ServoCheckWindow := FALSE;
END_IF

END_FUNCTION

// Objects/FB_Servo_V4_07/Helpers/F_ServoDirection
FUNCTION F_ServoDirection : MC_DIRECTION
VAR_INPUT
	ServoMoveType		: E_ServoMoveType;
END_VAR

CASE ServoMoveType OF
	eServoMoveType_MODULO_SHORTEST_PATH : 
		F_ServoDirection := MC_Shortest_Way;
	eServoMoveType_MODULO_POSITIVE : 
		F_ServoDirection := MC_Positive_Direction;
	eServoMoveType_MODULO_NEGATIVE : 
		F_ServoDirection := MC_Negative_Direction;
END_CASE

END_FUNCTION

// Objects/FB_Servo_V4_07/Helpers/F_ServoPositionCheck
FUNCTION F_ServoPositionCheck : BOOL
VAR_INPUT
	Unwind			: LREAL;
	MovePos			: REAL;
	ActualPos		: LREAL;
	PosTollerance	: REAL;
	Window			: REAL;
END_VAR
VAR
	Deviation		: LREAL;
END_VAR

IF (ActualPos < MovePos) THEN
	IF ABS((Unwind-MovePos)+ActualPos)<ABS(MovePos-ActualPos) THEN
		Deviation := -1* ((Unwind-MovePos)+ActualPos);
	ELSE
		Deviation := MovePos-ActualPos;
	END_IF
ELSE	
	IF ABS((Unwind-ActualPos)+MovePos)<ABS(ActualPos-MovePos) THEN
		Deviation :=  ((Unwind-ActualPos)+MovePos);
	ELSE
		Deviation := -1* (ActualPos-MovePos);
	END_IF
END_IF



F_ServoPositionCheck := ABS(Deviation) <= Window AND ABS(Deviation) > PosTollerance;

END_FUNCTION

// Objects/FB_Servo_V4_07/Helpers/FB_ServoMotionDynamics
FUNCTION_BLOCK FINAL FB_ServoMotionDynamics
VAR_INPUT
	ExecuteMove					: BOOL;				
END_VAR
VAR_IN_OUT
	Axis						: AXIS_REF;		
	CMD_Power					: MC_POWER;	
	BufferMode					: MC_BUFFERMODE;		
	PosMove1					: ST_MovePosition_SP;	
	CMD_MovePosAbs1				: MC_MOVEABSOLUTE;
	PosMove2					: ST_MovePosition_SP;	
	CMD_MovePosAbs2				: MC_MOVEABSOLUTE;
END_VAR
VAR
	_Reset						: MC_Reset;		
	_State						: E_MoveState;			
	_r_Trig						: R_TRIG;
END_VAR

//************************************************
//					CONTROL
//************************************************		

(* update the axis status at the beginning of each cycle *)
	Axis.ReadStatus();
	
	_r_Trig(CLK:= ExecuteMove);
	
	IF _r_Trig.Q THEN
		_State := MOVESTATE_ENABLE;
	END_IF

	(* move axis using a state machine *)
	CASE _State OF
		
		MOVESTATE_INIT :	(* initialisation *)
			(* initialize all function blocks *)
			CMD_MovePosAbs1.Execute := FALSE;
			CMD_MovePosAbs2.Execute := FALSE;
			_Reset.Execute := FALSE;

		MOVESTATE_ENABLE :

			IF CMD_Power.Status THEN
				_State := MOVESTATE_FORWARD;
			ELSIF CMD_Power.Error THEN
				_State := MOVESTATE_ERROR;
			END_IF

		MOVESTATE_FORWARD :		(* start to first position *)
			CMD_MovePosAbs1.BufferMode := MC_Buffered;
			CMD_MovePosAbs1.Execute := TRUE;
			IF CMD_MovePosAbs1.Active  THEN
				(* axis is executing job but is not yet finished *)
				CMD_MovePosAbs1.Execute := FALSE;
				(* leave this state and buffer a second command *)
				_State := MOVESTATE_NEWTARGETPOSITION;
			ELSIF CMD_MovePosAbs1.CommandAborted OR CMD_MovePosAbs1.Error THEN
				_State := MOVESTATE_ERROR;
			END_IF
			
		MOVESTATE_NEWTARGETPOSITION :(* change target position while moving *)
			CMD_MovePosAbs2.BufferMode := BufferMode; 	(* use velocity of previous command till intermediate target position position *)
			CMD_MovePosAbs2.Execute := TRUE;
			IF CMD_MovePosAbs2.Done THEN
				CMD_MovePosAbs2.Execute := FALSE;
				_State := MOVESTATE_INIT;
			ELSIF CMD_MovePosAbs2.CommandAborted OR CMD_MovePosAbs2.Error THEN
				_State := MOVESTATE_ERROR;
			END_IF

		MOVESTATE_ERROR :
			IF Axis.Status.Error THEN
				_State := MOVESTATE_RESET;	(* axis error requires reset *)
			ELSE
				_State := MOVESTATE_INIT;		(* function block errors don't need a reset *)
			END_IF

		MOVESTATE_RESET :
			_Reset.Execute := TRUE;
			IF _Reset.Done THEN
				_State := MOVESTATE_INIT;
			ELSIF _Reset.Error THEN
				_State := MOVESTATE_INIT; (* can't do anything here *)
			END_IF

	END_CASE
//************************************************
//					OUTPUTS
//************************************************	
	
_Reset(
	Axis:= Axis, 
	Execute:= , 
	Done=> , 
	Busy=> , 
	Error=> , 
	ErrorID=> );
	
CMD_MovePosAbs1(
	Axis:= Axis, 
	Execute:= , 
	Position:= PosMove1.Position, 
	Velocity:= PosMove1.Velocity, 
	Acceleration:= PosMove1.Acceleration, 
	Deceleration:= PosMove1.Deceleration, 
	Jerk:= PosMove1.Jerk, 
	BufferMode:= , 
	Options:= , 
	Done=> , 
	Busy=> , 
	Active=> , 
	CommandAborted=> , 
	Error=> , 
	ErrorID=> );
	
CMD_MovePosAbs2(
	Axis:= Axis, 
	Execute:= , 
	Position:= PosMove2.Position, 
	Velocity:= PosMove2.Velocity, 
	Acceleration:= PosMove2.Acceleration, 
	Deceleration:= PosMove2.Deceleration, 
	Jerk:= PosMove2.Jerk, 
	BufferMode:= , 
	Options:= , 
	Done=> , 
	Busy=> , 
	Active=> , 
	CommandAborted=> , 
	Error=> , 
	ErrorID=> );

END_FUNCTION_BLOCK

// Objects/FB_Servo_V4_07/Helpers/FB_ServoMove
FUNCTION_BLOCK FINAL FB_ServoMove
VAR_INPUT
	ExecuteMove					: BOOL;					
END_VAR
VAR_IN_OUT
	Axis						: AXIS_REF;				
	PosMove						: ST_MovePosition_SP;
	CMD_MovePosAbs				: MC_MOVEABSOLUTE;
	CMD_MovePosMod				: MC_MOVEMODULO;
	CMD_MovePosRel				: MC_MOVERELATIVE;	
END_VAR
VAR
	_accelRate					: LREAL;
	_decelRate					: LREAL;
	_jerkTime					: REAL;
	_jerkValue					: LREAL;
	_posMoveAbsActive			: BOOL;
	_posMoveRelActive			: BOOL;
	_posMoveModActive			: BOOL;
END_VAR

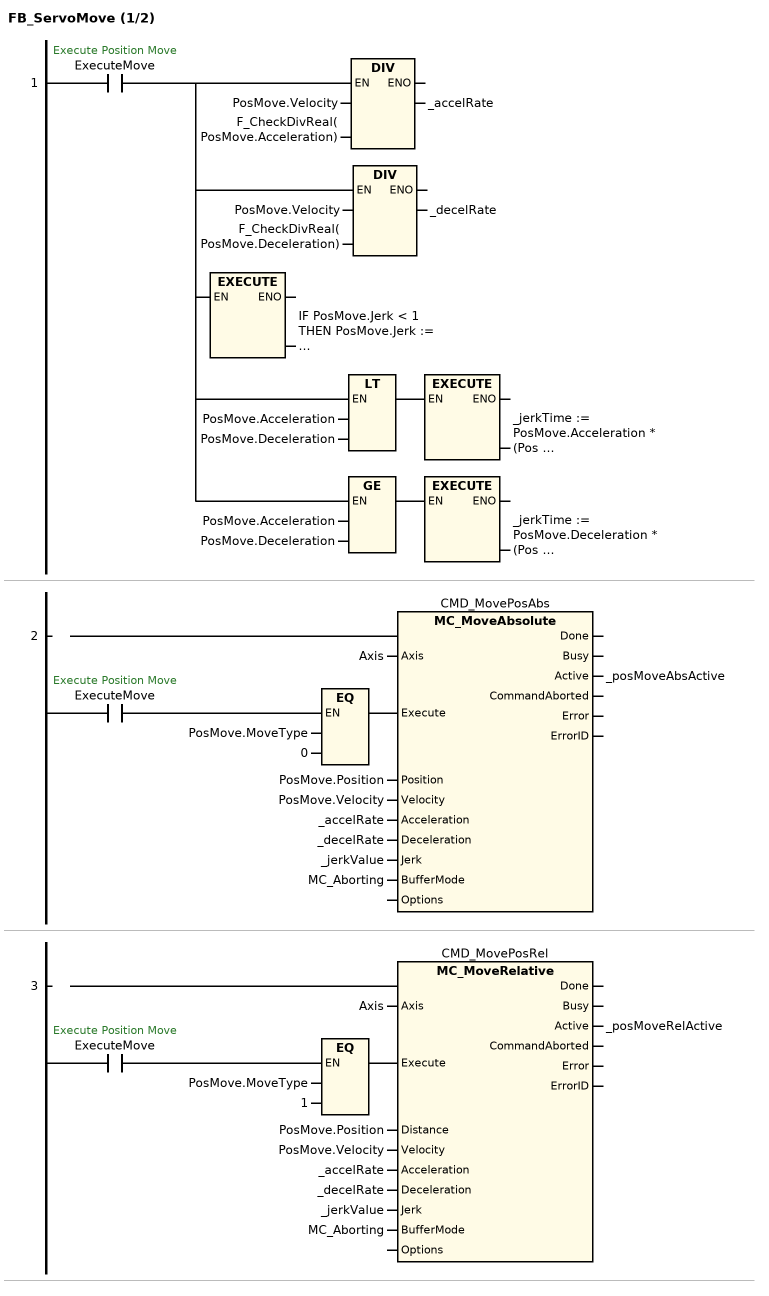
// NETWORK 1
//   ExecuteMove: Execute Position Move
//   PosMove.Velocity: Velocity Value of Move
//   F_CheckDivReal(PosMove.Acceleration): Accleration Value of Move
//   F_CheckDivReal(PosMove.Deceleration): Deceleration Value of Move
//   PosMove.Acceleration: Accleration Value of Move
//   PosMove.Deceleration: Deceleration Value of Move
IF ExecuteMove THEN _accelRate := PosMove.Velocity / (F_CheckDivReal(PosMove.Acceleration)); END_IF
IF ExecuteMove THEN _decelRate := PosMove.Velocity / (F_CheckDivReal(PosMove.Deceleration)); END_IF
IF ExecuteMove THEN
    IF PosMove.Jerk < 1 THEN PosMove.Jerk := 1; END_IF
    IF PosMove.Jerk > 100 THEN PosMove.Jerk := 100; END_IF
END_IF
IF ExecuteMove AND PosMove.Acceleration < PosMove.Deceleration THEN
    _jerkTime := PosMove.Acceleration * (PosMove.Jerk / 100);
    _jerkValue := _accelRate / F_CheckDivReal(_jerkTime);
END_IF
IF ExecuteMove AND PosMove.Acceleration >= PosMove.Deceleration THEN
    _jerkTime := PosMove.Deceleration * (PosMove.Jerk / 100);
    _jerkValue := _decelRate / F_CheckDivReal(_jerkTime);
END_IF

// NETWORK 2
//   ExecuteMove: Execute Position Move
//   PosMove.MoveType: Move Type Configuration of Positional Move
//   PosMove.Position: Position Value to Move to
//   PosMove.Velocity: Velocity Value of Move
CMD_MovePosAbs(
    Axis := Axis,
    Execute := ExecuteMove AND PosMove.MoveType = 0,
    Position := PosMove.Position,
    Velocity := PosMove.Velocity,
    Acceleration := _accelRate,
    Deceleration := _decelRate,
    Jerk := _jerkValue,
    BufferMode := MC_Aborting,
    Active => _posMoveAbsActive); // MC_MoveAbsolute

// NETWORK 3
//   ExecuteMove: Execute Position Move
//   PosMove.MoveType: Move Type Configuration of Positional Move
//   PosMove.Position: Position Value to Move to
//   PosMove.Velocity: Velocity Value of Move
CMD_MovePosRel(
    Axis := Axis,
    Execute := ExecuteMove AND PosMove.MoveType = 1,
    Distance := PosMove.Position,
    Velocity := PosMove.Velocity,
    Acceleration := _accelRate,
    Deceleration := _decelRate,
    Jerk := _jerkValue,
    BufferMode := MC_Aborting,
    Active => _posMoveRelActive); // MC_MoveRelative

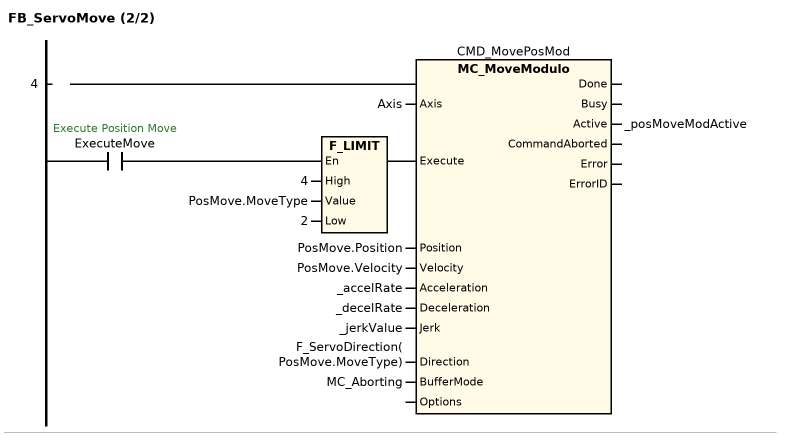
// NETWORK 4
//   ExecuteMove: Execute Position Move
//   PosMove.MoveType: Move Type Configuration of Positional Move
//   PosMove.Position: Position Value to Move to
//   PosMove.Velocity: Velocity Value of Move
CMD_MovePosMod(
    Axis := Axis,
    Execute := F_LIMIT(En := ExecuteMove, High := 4, Value := PosMove.MoveType, Low := 2),
    Position := PosMove.Position,
    Velocity := PosMove.Velocity,
    Acceleration := _accelRate,
    Deceleration := _decelRate,
    Jerk := _jerkValue,
    Direction := F_ServoDirection(PosMove.MoveType),
    BufferMode := MC_Aborting,
    Active => _posMoveModActive); // MC_MoveModulo

END_FUNCTION_BLOCK

// Objects/FB_Servo_V4_07/FB_Servo
FUNCTION_BLOCK FINAL FB_Servo EXTENDS FB_EventLogger
VAR_INPUT
	Energized 							: BOOL;	
	Disable								: BOOL;				
	HomingInput							: BOOL;
	EnableMoves							: BOOL;
	EnableMotionDynamics				: BOOL;
	EnableContinousRun					: BOOL;
	EnableSuperImpose					: BOOL;
	EnableCamming						: BOOL;
	Virtual								: BOOL;			
END_VAR                     			
VAR_IN_OUT	                			
	Master								: AXIS_REF;
	Control								: ST_System;				
END_VAR                     			
VAR_OUTPUT                  												
	StepNum								: DINT;				
END_VAR      
VAR PERSISTENT                      	
	_Name								: STRING[15];						//Name for HMI
	_Description						: STRING[40];						//Description for HMI
	_AlarmMute							: BOOL;								//Alarm Mute
	_FaultTimer_PT						: REAL;								//Fault timer preset time	
	_PosSyncMove						: ST_MovePosition_SP;				//Sync Position Move Setpoints
	_PosMove							: ARRAY[1..4] OF ST_MovePosition_SP;//Position Move Setpoints
	_PosMoveDynamicsStart				: ARRAY[1..4] OF ST_MovePosition_SP;//Motion Dynamic Start Position Move Setpoints
	_PosMoveDynamicsEnd					: ARRAY[1..4] OF ST_MovePosition_SP;//Motion Dynamic End Position Move Setpoints
	_MD_BufferMode						: ARRAY[1..4] OF MC_BUFFERMODE;		//Motion Dynamic BufferMode for successive travel commands.
	_MoveSuperImposed					: ST_MoveSuperImposed_SP;			//Starts a relative superimposed movement while the axis is already moving
	_PosMoveHome						: ST_HomePosition_SP;				//Position Data for Homing
	_PosMoveHaltDec						: REAL;								//Positional Move Halt Deceration
	_PosMoveHaltJerk					: REAL;								//Positional Move Halt Jerk
	_ManualPositionMove					: ST_MovePosition_SP;				//Manual Position Move Setpoints
	_Jog								: ST_ConstantVelocity_SP;			//Jog Setpoints
	_ContinuousRun						: ST_ConstantVelocity_SP;			//Continuous Run Setpoints
	_EStopDec							: REAL := 95;						//EStop Deceleration Percentage
	_Settings							: ST_Settings_SP;					//Drive Parameters
	_DriveRef							: ST_DriveRef;						//Drive Reference Access
	_RunHours							: REAL;								//Total hours the servo has run
	_Homed								: BOOL;								//Servo is Homed
	_HomeMode							: INT;								//Home Mode 0:=Backwards then Forwards 1:=Forwards then Forwards, 2:= Forwards then Backwards, 3:= Set Position, 4:= Set Position Offset
	_HomingTorqueLimit					: UINT := 20;						//Homing Torque Limit
	_NormalTorqueLimit					: UINT := 50;						//Normal Torque Limit (%)
	_NormalTorqueLimitNm				: LREAL;							//Normal Torque Limit (nM)
	_CamTable							: ST_CamTable; 						//Cam table
	_Unit								: STRING(8);						//Servo Position Unit, i.e deg, mm etc
	_ServoTorqueLimit  		AT %Q*		: UINT;			    				//S-0-0092: Bipolar torque/force limit value    
	_MaxDriveOffDelay					: DINT;								//S-0-0273: Maximum drive off delay (ms)
	_MaxDriveOffDelayWrite				: DINT;								//S-0-0273: Maximum drive off delay (ms) write variable for testing
	_MotorPeakForce						: REAL;								//P-0-0128: Motor peak force
	_Variables							: ARRAY [0..9] OF ST_Variable;		//Device Associated Varibles Array		
END_VAR                       	
VAR                                 	
	_Axis								: AXIS_REF;							//Axis Reference
	_DriveStatus			 			: ST_AX5000DriveStatus;				//Drive Status 
	_ExtControl							: BOOL;								//To be Enabled if used in conjunction with another AOI E.g Kinematics 2D
	_ExtManEn							: BOOL;								//For External Manual Control
	_AutoEn								: BOOL;								//Auto Enable
	_ManPos								: BOOL;								//Jog Positive
	_ManNeg								: BOOL;								//Jog Negative
	_ManPosition						: BOOL;								//Jog to Manual Setpoint
	_ForcePos							: BOOL;								//Jog Positive
	_ForceNeg							: BOOL;								//Jog Negative
	_ForceOff							: BOOL;								//Manual Off
	_ManOff								: BOOL;								//Manual Off
	_AutoHome							: BOOL;								//Command Home Drive Auto
	_MovePosSync						: BOOL;								//Command to Move the the Cam Sync Position
	_PosSyncOK							: BOOL;								//Servo is in Sync Position
	_MovePos							: ARRAY[1..4] OF BOOL;				//Command to move to Position
	_PosOK								: ARRAY[1..4] OF BOOL;      		//Servo is in Position
	_MoveDynamic						: ARRAY[1..4] OF BOOL;	    		//Command motion dynamic move to Position 
	_PosDynamicOK						: ARRAY[1..4] OF BOOL;				//Servo is in Motion Dynamic Position 
	_MoveHalt							: BOOL;								//Command Stop Move In Progress
	_ContRun							: BOOL;								//Start Continuous Run
	_MoveSuperImpose					: BOOL;								//Start a super impose move
	_UpdateDriveParameters				: BOOL;								//Command Update Drive Parameters
	_ManHome							: ST_Selection;						//Command Home Drive Manual
	_RunCam								: BOOL;								//Command to Run Cam Profile
	_ManBrakeRelease					: BOOL;								//Manual Brake Release
	_Enabled							: BOOL;								//Servo is Enabled
	_HomeSeqStep						: STRING;							//Homing Sequence Step String
	_StandStill							: BOOL;								//Servo is not Moving
	_Fault								: BOOL;	     						//Device Fault
	_FaultTimer_ET						: REAL;								//Fault timer elapsed
	_ManualJogActive					: BOOL;								//Servo is Manual Jogging
	_ManualMoveActive					: BOOL;								//Servo is Manual Moving
	_MaximumDeceleration				: LREAL;							//Maximum Deceleration of the System
	_Moving								: BOOL;								//Servo is currently moving
	_MoveTime							: REAL;								//Time servo has been moving (seconds)
	_CamInSync							: BOOL;								//Servo cam coupling was successful
	_Alarm								: BOOL;								//Device Alarm         
	_Warning							: BOOL;								//Device Warning          
	_AlarmNum							: UDINT;							//Device Alarm Number  
	_WarningNum							: DINT;								//Device Warning Number
	_DigitalInputs    		AT %I*  	: INT;								//P-0-0801: Digital Inputs
	_DriveStatusWord   		AT %I*		: WORD;								//S-0-0135: Drive Status Word
	_SafetyOptionState 					: WORD;								//P-0-2002: Safety Option State
	_SafetyStateBool					: BOOL;								//P-0-2002 is a word, safety state bool represents bool state
	_TorqueCurrent     		AT %I*		: INT;			    				//P-0-0459: Actual torque/force generating current
	_TorqueFeedbackPercent				: INT;			    				//S-0-0084: Torque/force feedback  
	_TorquePeak							: DINT;								//P-0-0094
	_TorqueFeedback						: LREAL;							//Torque Feedback from Drive
	{attribute 'tc_no_symbol'}	
	_ActMotorBreakCurrentRead			: INT;								//P-0-0064: Actual Motor
	_ActMotorBreakCurrent				: REAL;								//P-0-0064: Actual Motor Break Current           
	_ManEN								: BOOL;								//Manual Control Enabled
	_HomingEN							: BOOL;								//Homing Enabled
	_Step								: DWORD;							//Servo Control Step
	{attribute 'tc_no_symbol'}                	                			
	_CMD_SoEReset						: FB_SoEReset;						//Axis Reset Command
	{attribute 'tc_no_symbol'}                	                			
	_CMD_Power							: MC_POWER;							//Power Axis Command
END_VAR

_Axis.ReadStatus();
M_UnlatchManuals();
M_StateControl();
M_StateOutputs();
M_Homing();
M_Jogging();
M_ControlOutputs();
M_SettingsControl();
M_WarningMonitor();
M_AlarmMonitor();
M_BrakeControl();
M_GetDiagnosis();

//Enable Functions
IF EnableMoves THEN M_MoveToPosition(); END_IF
IF EnableMotionDynamics	THEN M_MotionDynamicMove(); END_IF
IF EnableContinousRun THEN M_ContinuousRun(); END_IF
IF EnableSuperImpose THEN M_MoveSuperImposed(); END_IF
//IF EnableCamming THEN M_Camming(); END_IF

//Run hours
IF Control.Inputs.HoursReset THEN
	_RunHours := 0;
END_IF
IF _Axis.Status.Moving AND NOT Control.Inputs.HoursReset THEN
	_Moving := TRUE;
	_RunHours := _RunHours + (Control.SystemTime.ScanTime/3600);
	_MoveTime := _MoveTime + Control.SystemTime.ScanTime;
ELSE
	_Moving := FALSE;
	_MoveTime := 0;
END_IF

{attribute 'monitoring' := 'variable'}
PROPERTY PUBLIC Alarm : Bool
GET
Alarm := _Alarm;
END_GET
END_PROPERTY

{attribute 'monitoring' := 'variable'}
PROPERTY PUBLIC AlarmMute : BOOL
SET
AlarmMute := _AlarmMute;
END_SET
END_PROPERTY

{attribute 'monitoring' := 'variable'}
PROPERTY PUBLIC AutoEn : Bool
GET
AutoEn := _AutoEn;
END_GET
SET
_AutoEn := AutoEn;
END_SET
END_PROPERTY

{attribute 'monitoring' := 'variable'}
PROPERTY PUBLIC AutoHome : Bool
GET
AutoHome := _AutoHome;
END_GET
SET
_AutoHome := AutoHome;
END_SET
END_PROPERTY

{attribute 'monitoring' := 'variable'}
PROPERTY PUBLIC AxisEnabled : Bool
GET
AxisEnabled := _Enabled;
END_GET
END_PROPERTY

{attribute 'monitoring' := 'variable'}
PROPERTY PUBLIC CamInSync : Bool
GET
CamInSync := _CamInSync;
END_GET
END_PROPERTY

{attribute 'Suspress_wrn_C0410'}
PROPERTY PUBLIC ContinuousRun : REFERENCE TO ST_ConstantVelocity_SP
GET
PUBLIC 
VAR
END_VAR
ContinuousRun REF= _ContinuousRun;
END_GET
SET
_ContinuousRun := ContinuousRun;
END_SET
END_PROPERTY

{attribute 'monitoring' := 'variable'}
PROPERTY PUBLIC ContRun : Bool
SET
_ContRun := ContRun;
END_SET
END_PROPERTY

{attribute 'monitoring' := 'variable'}
PROPERTY PUBLIC Description : String[40]
GET
Description := _Description;
END_GET
SET
_Description := Description;
END_SET
END_PROPERTY

{attribute 'monitoring' := 'variable'}
PROPERTY PUBLIC DigitalInputs : INT
GET
DigitalInputs := _DigitalInputs;
END_GET
SET
_DigitalInputs := DigitalInputs;
END_SET
END_PROPERTY

{attribute 'monitoring' := 'variable'}
PROPERTY PUBLIC ExtControl : Bool
SET
_ExtControl := ExtControl;
END_SET
END_PROPERTY

{attribute 'monitoring' := 'variable'}
PROPERTY PUBLIC ExtManEn : Bool
SET
_ExtManEn := ExtManEn;
END_SET
END_PROPERTY

{attribute 'monitoring' := 'variable'}
PROPERTY PUBLIC Fault : Bool
SET
_Fault := Fault;
END_SET
END_PROPERTY

{attribute 'monitoring' := 'variable'}
PROPERTY PUBLIC FaultTimer_ET : real
GET
FaultTimer_ET := _FaultTimer_ET;
END_GET
END_PROPERTY

{attribute 'monitoring' := 'variable'}
PROPERTY PUBLIC FaultTimer_PT : real
GET
FaultTimer_PT := _FaultTimer_PT;
END_GET
SET
_FaultTimer_PT := FaultTimer_PT;
END_SET
END_PROPERTY

{attribute 'monitoring' := 'variable'}
PROPERTY PUBLIC ForceNeg : Bool
GET
ForceNeg := _ForceNeg;
END_GET
SET
_ForceNeg := ForceNeg;
END_SET
END_PROPERTY

{attribute 'monitoring' := 'variable'}
PROPERTY PUBLIC ForcePos : Bool
GET
ForcePos := _ForcePos;
END_GET
SET
_ForcePos := ForcePos;
END_SET
END_PROPERTY

{attribute 'monitoring' := 'variable'}
PROPERTY PUBLIC Homed : Bool
GET
Homed := _Homed;
END_GET
END_PROPERTY

{attribute 'monitoring' := 'variable'}
PROPERTY PUBLIC HomeMode : INT
GET
HomeMode := _HomeMode;
END_GET
SET
_HomeMode := HomeMode;
END_SET
END_PROPERTY

{attribute 'monitoring' := 'variable'}
PROPERTY PUBLIC Jog : REFERENCE TO ST_ConstantVelocity_SP
GET
Jog REF= _Jog;
END_GET
SET
_Jog := Jog;
END_SET
END_PROPERTY

METHOD PRIVATE M_AlarmMonitor
VAR_INPUT
END_VAR
VAR_INST
	{attribute 'tc_no_symbol'}                	                			
	_R_Trig				:   ARRAY[0..2] OF R_TRIG;		
END_VAR
IF NOT _AlarmMute AND NOT Control.Inputs.AlarmAck.Enabled  THEN

	_R_Trig[0](CLK:= _Fault);
	_R_Trig[1](CLK:= _Axis.NcToPlc.ErrorCode <> 0);	
	_R_Trig[2](CLK:= _Axis.Status.ErrorStop OR _Axis.Status.Error);	

	IF _Fault THEN
		_FaultTimer_ET := _FaultTimer_ET + Control.SystemTime.ScanTime;
		IF _R_Trig[0].Q THEN
			_FaultTimer_ET := 0;
		ELSIF _FaultTimer_ET > _FaultTimer_PT THEN
			_AlarmNum := 1101;
		END_IF
	ELSIF _R_Trig[1].Q THEN
		_AlarmNum := _Axis.Status.ErrorID;
	ELSIF _R_Trig[2].Q THEN 
		_AlarmNum := _Axis.NcToPlc.ErrorCode;					
	END_IF
		
	IF _AlarmNum <> 0 THEN 	
		_Alarm := TRUE;
		IF NOT Control.Outputs.Alarm THEN
			Control.Outputs.Alarm := TRUE;
		END_IF
	ELSE
		_Alarm := FALSE;
	END_IF
	
END_IF

IF Control.Inputs.AlarmAck.Enabled OR _AlarmMute THEN
	_AlarmNum:=0;
	_FaultTimer_ET := 0;
END_IF

M_LogAlarm(
	Execute:= _Alarm, 
	Arg0:= _Name, 
	Arg1:= _Description, 
	Arg2:= M_Errors(), 
	Clear:= NOT _Alarm, 
	EventEntry:= M_Alarms(), 
	Message:= Control.Outputs.AlarmMessage);
END_METHOD

METHOD PRIVATE M_Alarms : TcEventEntry
VAR_INPUT
END_VAR
VAR_INST
END_VAR
CASE _AlarmNum OF
	1101:    M_Alarms := TC_Events.TcServo.A_1101;//Alarm			
ELSE
	IF _AlarmNum >= 16384 AND _AlarmNum <= 16497 THEN
		M_Alarms := TC_Events.TcServo.A_1102;//General Errors
	ELSIF _AlarmNum >= 16641 AND _AlarmNum <= 16756 THEN
		M_Alarms := TC_Events.TcServo.A_1103;//Channel Errors
	ELSIF _AlarmNum >= 16896 AND _AlarmNum <= 17151 THEN
		M_Alarms := TC_Events.TcServo.A_1104;//Group Errors
	ELSIF _AlarmNum >= 17152 AND _AlarmNum <= 17312 THEN
		M_Alarms := TC_Events.TcServo.A_1105;//Axis Errors
	ELSIF _AlarmNum >= 17408 AND _AlarmNum <= 17571 THEN
		M_Alarms := TC_Events.TcServo.A_1106;//Encoder Errors
	ELSIF _AlarmNum >= 17664 AND _AlarmNum <= 17828 THEN
		M_Alarms := TC_Events.TcServo.A_1107;//Controller Errors
	ELSIF _AlarmNum >= 17920 AND _AlarmNum <= 18005 THEN
		M_Alarms := TC_Events.TcServo.A_1108;//Drive Errors
	ELSIF _AlarmNum >= 18944 AND _AlarmNum <= 18979 THEN
		M_Alarms := TC_Events.TcServo.A_1109;//Table Errors
	ELSIF _AlarmNum >= 19200 AND _AlarmNum <= 19383 THEN
		M_Alarms := TC_Events.TcServo.A_1110;//NC-PLC Errors
	ELSIF _AlarmNum >= 19456 AND _AlarmNum <= 19536 THEN
		M_Alarms := TC_Events.TcServo.A_1111;//Kinematic transformation Errors
	ELSIF _AlarmNum >= 33024 AND _AlarmNum <= 33042 THEN
		M_Alarms := TC_Events.TcServo.A_1112;//Bode Return Codes
	ELSIF _AlarmNum >= 33056 AND _AlarmNum <= 33136 THEN
		M_Alarms := TC_Events.TcServo.A_1113;//Further Error Codes
	ELSIF _AlarmNum >= 1 AND _AlarmNum <= 30 THEN
		M_Alarms := TC_Events.TcServo.A_1114;//Global error codes
	ELSIF _AlarmNum >= 1280 AND _AlarmNum <= 1293 THEN
		M_Alarms := TC_Events.TcServo.A_1115;//Router error codes
	ELSIF _AlarmNum >= 1792 AND _AlarmNum <= 1877 THEN
		M_Alarms := TC_Events.TcServo.A_1116;//General ADS error codes
	ELSIF _AlarmNum >= 4096 AND _AlarmNum <= 4122 THEN
		M_Alarms := TC_Events.TcServo.A_1117;//RTime error codes
	ELSIF _AlarmNum >= 10060 AND _AlarmNum <= 10065 THEN
		M_Alarms := TC_Events.TcServo.A_1118;//TCP Winsock error codes
	ELSE
		M_Alarms := TC_Events.TcServo.A_Undefined;
	END_IF

END_CASE
END_METHOD

METHOD M_BrakeControl
VAR_INST
	{attribute 'tc_no_symbol'}                	                			
	_CMD_BrakeRelease		: FB_SoEAX5000SetMotorCtrlWord;	
	{attribute 'tc_no_symbol'}                	                			
	_CMD_BrakeAuto			: FB_SoEAX5000SetMotorCtrlWord;		
END_VAR
VAR_INST // added by the converter: edge detectors and wires of the graphical bodies
    _rt1, _rt2, _rt3 : R_TRIG;
    _w1, _w2 : BOOL;
    _ft1 : F_TRIG;
END_VAR
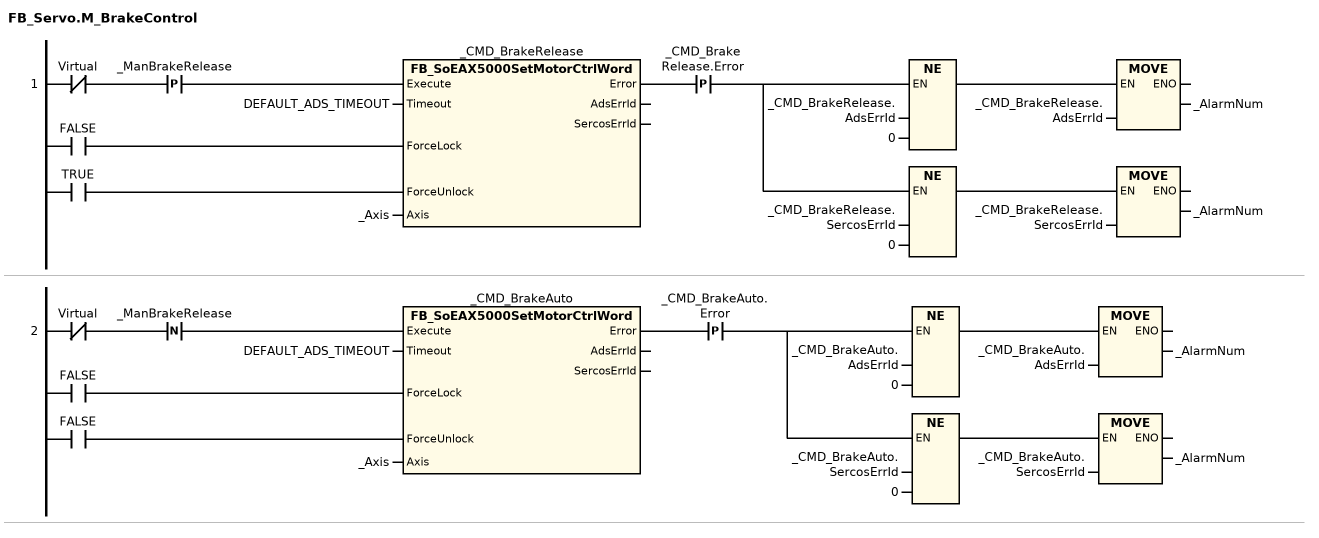
// NETWORK 1
_rt1(CLK := _ManBrakeRelease);
_CMD_BrakeRelease(
    Execute := NOT Virtual AND _rt1.Q,
    Timeout := DEFAULT_ADS_TIMEOUT,
    ForceLock := FALSE,
    ForceUnlock := TRUE,
    Axis := _Axis); // FB_SoEAX5000SetMotorCtrlWord
_rt2(CLK := _CMD_BrakeRelease.Error);
_w1 := _CMD_BrakeRelease.Error AND _rt2.Q;
IF _w1 AND _CMD_BrakeRelease.AdsErrId <> 0 THEN _AlarmNum := _CMD_BrakeRelease.AdsErrId; END_IF
IF _w1 AND _CMD_BrakeRelease.SercosErrId <> 0 THEN _AlarmNum := _CMD_BrakeRelease.SercosErrId; END_IF

// NETWORK 2
_ft1(CLK := _ManBrakeRelease);
_CMD_BrakeAuto(
    Execute := NOT Virtual AND _ft1.Q,
    Timeout := DEFAULT_ADS_TIMEOUT,
    ForceLock := FALSE,
    ForceUnlock := FALSE,
    Axis := _Axis); // FB_SoEAX5000SetMotorCtrlWord
_rt3(CLK := _CMD_BrakeAuto.Error);
_w2 := _CMD_BrakeAuto.Error AND _rt3.Q;
IF _w2 AND _CMD_BrakeAuto.AdsErrId <> 0 THEN _AlarmNum := _CMD_BrakeAuto.AdsErrId; END_IF
IF _w2 AND _CMD_BrakeAuto.SercosErrId <> 0 THEN _AlarmNum := _CMD_BrakeAuto.SercosErrId; END_IF
END_METHOD

METHOD PRIVATE M_ContinuousRun
VAR_INPUT
END_VAR
VAR_INST
	{attribute 'tc_no_symbol'}                	                			
	_CMD_ContinuousRun					: MC_MOVEVELOCITY;
	{attribute 'tc_no_symbol'}                	                			
	_CMD_ContinuousRunStop				: MC_STOP;
	{attribute 'tc_no_symbol'}                	                			
	_Step								: SINT;
	{attribute 'tc_no_symbol'} 	
	_R_Trig								: ARRAY[0..2] OF R_TRIG;
	{attribute 'tc_no_symbol'}                	                			
	_jerkValue							: LREAL;
	{attribute 'tc_no_symbol'}                	                			
	_jerkTime							: LREAL;
END_VAR
IF _ContinuousRun.Jerk < 1 THEN _ContinuousRun.Jerk := 1; END_IF
IF _ContinuousRun.Jerk > 100 THEN _ContinuousRun.Jerk := 100; END_IF

IF _ContinuousRun.Acceleration < _ContinuousRun.Deceleration THEN 
	_jerkTime := _ContinuousRun.Acceleration * (_ContinuousRun.Jerk / 100);
	IF _jerkTime > 0 THEN
		_jerkValue := _ContinuousRun.Velocity/F_CheckDivReal(_ContinuousRun.Acceleration) / F_CheckDivReal(LREAL_TO_REAL(_jerkTime));
	END_IF
ELSE
	_jerkTime := _ContinuousRun.Deceleration * (_ContinuousRun.Jerk / 100);
	IF _jerkTime > 0 THEN
		_jerkValue := _ContinuousRun.Velocity/F_CheckDivReal(_ContinuousRun.Deceleration) / F_CheckDivReal(LREAL_TO_REAL(_jerkTime));
	END_IF
END_IF

_CMD_ContinuousRun(
	Axis:= _Axis, 
	Velocity:=_ContinuousRun.Velocity , 
	Acceleration:= _ContinuousRun.Velocity/F_CheckDivReal(_ContinuousRun.Acceleration), 
	Deceleration:= _ContinuousRun.Velocity/F_CheckDivReal(_ContinuousRun.Deceleration), 
	Jerk:= _jerkValue, 
	Direction:= _ContinuousRun.Direction, 
	BufferMode:=MC_Aborting );
	
_R_Trig[0](CLK:=_CMD_ContinuousRun.Error);IF _R_Trig[0].Q THEN _AlarmNum := _CMD_ContinuousRun.ErrorID; END_IF
	
_CMD_ContinuousRunStop(
	Axis:=  _Axis,  
	Deceleration:=  _ContinuousRun.Velocity/F_CheckDivReal(_ContinuousRun.Deceleration), 
	Jerk:= _jerkValue);
	
_R_Trig[1](CLK:=_CMD_ContinuousRunStop.Error);IF _R_Trig[1].Q THEN _AlarmNum := _CMD_ContinuousRunStop.ErrorID; END_IF

_R_Trig[2](CLK:=_Homed);IF _R_Trig[2].Q THEN _Step := 0; END_IF

CASE _Step OF
	
0:
	_CMD_ContinuousRun.Execute := FALSE;
	IF  _Enabled AND _ContRun THEN
		 _Step := 1;
	END_IF
1:
	_CMD_ContinuousRun.Execute := TRUE;
	IF  NOT _ContRun AND _Enabled THEN
		_Step := 2;
	ELSIF NOT _Enabled THEN
		_Step := 0;
	END_IF
2:
	_CMD_ContinuousRun.Execute := FALSE;
	IF  NOT _CMD_ContinuousRun.Busy THEN
		 _Step := 3;
	END_IF

3:
	_CMD_ContinuousRunStop.Execute := TRUE;
	IF  _CMD_ContinuousRunStop.Busy THEN
		 _Step := 4;
	END_IF

4:
	_CMD_ContinuousRunStop.Execute := FALSE;
		IF  NOT _CMD_ContinuousRunStop.Busy THEN
		 _Step := 0;
	END_IF

END_CASE
END_METHOD

METHOD PRIVATE M_ControlOutputs
VAR_INPUT
END_VAR
VAR_INST
END_VAR
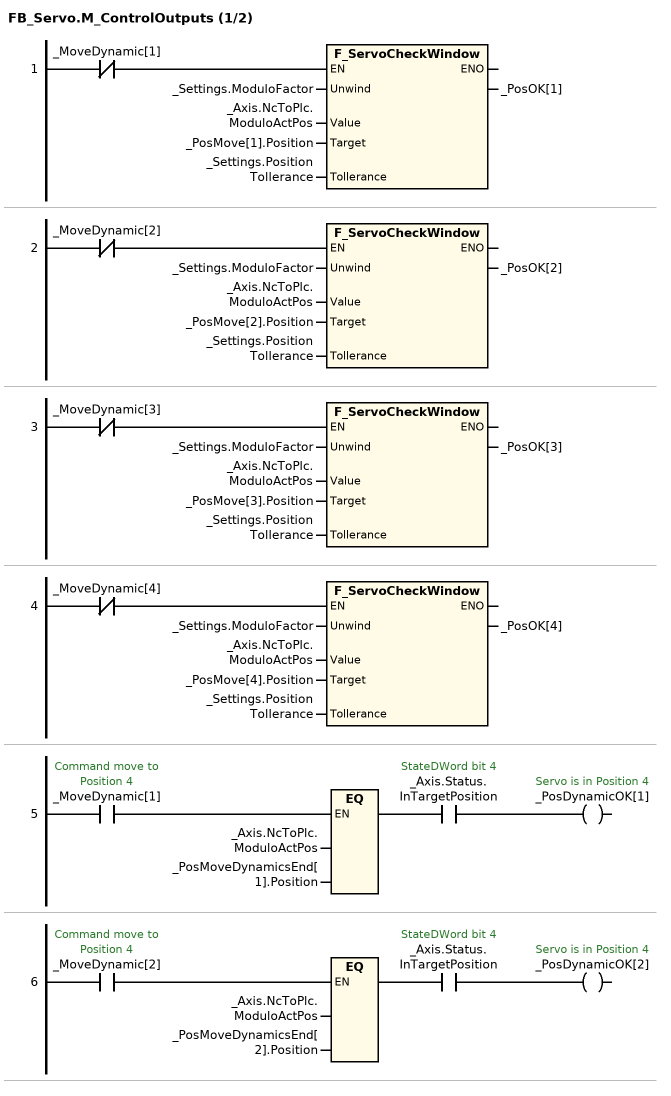
// NETWORK 1
IF NOT _MoveDynamic[1] THEN
    _PosOK[1] := F_ServoCheckWindow(Unwind := _Settings.ModuloFactor, Value := _Axis.NcToPlc.ModuloActPos, Target := _PosMove[1].Position, Tollerance := _Settings.PositionTollerance);
END_IF

// NETWORK 2
IF NOT _MoveDynamic[2] THEN
    _PosOK[2] := F_ServoCheckWindow(Unwind := _Settings.ModuloFactor, Value := _Axis.NcToPlc.ModuloActPos, Target := _PosMove[2].Position, Tollerance := _Settings.PositionTollerance);
END_IF

// NETWORK 3
IF NOT _MoveDynamic[3] THEN
    _PosOK[3] := F_ServoCheckWindow(Unwind := _Settings.ModuloFactor, Value := _Axis.NcToPlc.ModuloActPos, Target := _PosMove[3].Position, Tollerance := _Settings.PositionTollerance);
END_IF

// NETWORK 4
IF NOT _MoveDynamic[4] THEN
    _PosOK[4] := F_ServoCheckWindow(Unwind := _Settings.ModuloFactor, Value := _Axis.NcToPlc.ModuloActPos, Target := _PosMove[4].Position, Tollerance := _Settings.PositionTollerance);
END_IF

// NETWORK 5
//   _MoveDynamic[1]: Command move to Position 4
//   _PosMoveDynamicsEnd[1].Position: Position Value to Move to
//   _Axis.Status.InTargetPosition: StateDWord bit 4
//   _PosDynamicOK[1]: Servo is in Position 4
_PosDynamicOK[1] := (_MoveDynamic[1] AND _Axis.NcToPlc.ModuloActPos = _PosMoveDynamicsEnd[1].Position) AND _Axis.Status.InTargetPosition;

// NETWORK 6
//   _MoveDynamic[2]: Command move to Position 4
//   _PosMoveDynamicsEnd[2].Position: Position Value to Move to
//   _Axis.Status.InTargetPosition: StateDWord bit 4
//   _PosDynamicOK[2]: Servo is in Position 4
_PosDynamicOK[2] := (_MoveDynamic[2] AND _Axis.NcToPlc.ModuloActPos = _PosMoveDynamicsEnd[2].Position) AND _Axis.Status.InTargetPosition;

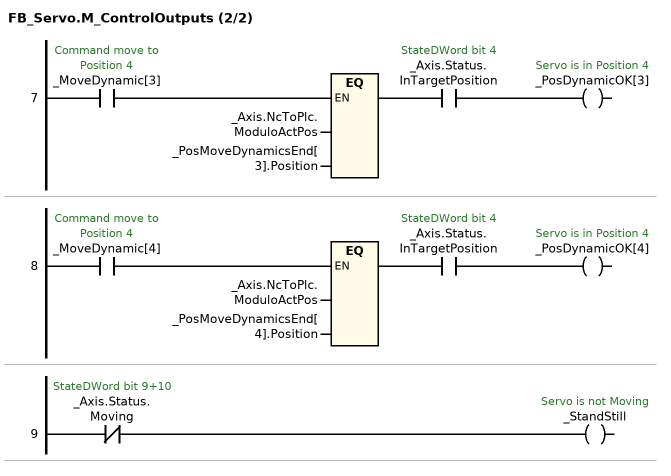
// NETWORK 7
//   _MoveDynamic[3]: Command move to Position 4
//   _PosMoveDynamicsEnd[3].Position: Position Value to Move to
//   _Axis.Status.InTargetPosition: StateDWord bit 4
//   _PosDynamicOK[3]: Servo is in Position 4
_PosDynamicOK[3] := (_MoveDynamic[3] AND _Axis.NcToPlc.ModuloActPos = _PosMoveDynamicsEnd[3].Position) AND _Axis.Status.InTargetPosition;

// NETWORK 8
//   _MoveDynamic[4]: Command move to Position 4
//   _PosMoveDynamicsEnd[4].Position: Position Value to Move to
//   _Axis.Status.InTargetPosition: StateDWord bit 4
//   _PosDynamicOK[4]: Servo is in Position 4
_PosDynamicOK[4] := (_MoveDynamic[4] AND _Axis.NcToPlc.ModuloActPos = _PosMoveDynamicsEnd[4].Position) AND _Axis.Status.InTargetPosition;

// NETWORK 9
//   _Axis.Status.Moving: StateDWord bit 9+10
//   _StandStill: Servo is not Moving
_StandStill := NOT _Axis.Status.Moving;
END_METHOD

